C07159=1025.520,281.444,-127.927,170.391,47.586,159.168
C07160=1025.514,281.195,-127.896,170.386,47.588,159.168
C07161=1025.507,280.947,-127.864,170.382,47.590,159.168
C07162=1025.501,280.699,-127.834,170.378,47.592,159.168
C07163=1025.495,280.452,-127.803,170.374,47.594,159.168
C07164=1025.487,280.204,-127.772,170.369,47.596,159.167
C07165=1025.481,279.956,-127.741,170.364,47.598,159.167
C07166=1025.474,279.708,-127.710,170.361,47.600,159.167
C07167=1025.468,279.459,-127.679,170.356,47.602,159.167
C07168=1025.461,279.212,-127.648,170.352,47.604,159.167
C07169=1025.455,278.963,-127.617,170.347,47.606,159.167
C07170=1025.448,278.716,-127.586,170.343,47.608,159.167
C07171=1025.437,278.308,-127.536,170.336,47.611,159.166
C07172=1025.427,277.900,-127.485,170.329,47.615,159.166
C07173=1025.416,277.492,-127.434,170.322,47.618,159.166
C07174=1025.405,277.084,-127.384,170.315,47.621,159.166
C07175=1025.399,276.836,-127.353,170.311,47.623,159.166
C07176=1025.392,276.588,-127.322,170.306,47.625,159.166
C07177=1025.385,276.340,-127.292,170.302,47.627,159.166
C07178=1025.379,276.092,-127.261,170.298,47.630,159.166
C07179=1025.372,275.843,-127.231,170.294,47.632,159.165
C07180=1025.366,275.596,-127.200,170.290,47.634,159.165
C07181=1025.359,275.348,-127.170,170.286,47.636,159.165
C07182=1025.352,275.100,-127.139,170.281,47.638,159.165
C07183=1025.346,274.852,-127.109,170.277,47.640,159.165
C07184=1025.339,274.604,-127.079,170.272,47.642,159.165
C07185=1025.333,274.356,-127.049,170.269,47.645,159.165
C07186=1025.326,274.108,-127.018,170.264,47.647,159.165
C07187=1025.319,273.860,-126.987,170.259,47.649,159.165
C07188=1025.314,273.612,-126.957,170.256,47.651,159.165
C07189=1025.306,273.364,-126.927,170.251,47.653,159.165
C07190=1025.300,273.115,-126.896,170.248,47.655,159.164
C07191=1025.293,272.868,-126.866,170.243,47.658,159.164
C07192=1025.287,272.619,-126.835,170.239,47.659,159.164
C07193=1025.280,272.371,-126.806,170.235,47.662,159.164
C07194=1025.274,272.123,-126.775,170.230,47.664,159.164
C07195=1025.267,271.875,-126.745,170.227,47.666,159.164
C07196=1025.261,271.627,-126.714,170.222,47.669,159.164
C07197=1025.254,271.379,-126.684,170.218,47.670,159.164
C07198=1025.248,271.131,-126.654,170.214,47.673,159.164
C07199=1025.241,270.883,-126.624,170.209,47.675,159.164
C07200=1025.235,270.635,-126.594,170.206,47.678,159.164
C07201=1025.228,270.387,-126.563,170.201,47.680,159.164
C07202=1025.222,270.139,-126.533,170.198,47.682,159.164
C07203=1025.215,269.891,-126.503,170.193,47.684,159.164
C07204=1025.208,269.643,-126.473,170.190,47.687,159.164
C07205=1025.202,269.394,-126.443,170.185,47.689,159.164
C07206=1025.196,269.146,-126.413,170.182,47.691,159.164
C07207=1025.189,268.898,-126.383,170.177,47.693,159.163
C07208=1025.183,268.650,-126.353,170.172,47.696,159.163
C07209=1025.176,268.402,-126.323,170.169,47.698,159.164
C07210=1025.169,268.154,-126.294,170.164,47.700,159.163
C07211=1025.163,267.906,-126.263,170.161,47.703,159.163
C07212=1025.156,267.658,-126.233,170.156,47.705,159.163
C07213=1025.150,267.409,-126.204,170.153,47.707,159.163
C07214=1025.144,267.161,-126.174,170.148,47.710,159.163
C07215=1025.137,266.913,-126.143,170.144,47.712,159.163
C07216=1025.130,266.666,-126.114,170.140,47.715,159.163
C07217=1025.124,266.417,-126.084,170.136,47.717,159.163
C07218=1025.117,266.169,-126.054,170.132,47.719,159.163
C07219=1025.110,265.920,-126.025,170.128,47.722,159.163
C07220=1025.104,265.673,-125.995,170.124,47.724,159.163
C07221=1025.097,265.425,-125.965,170.120,47.727,159.163
C07222=1025.091,265.176,-125.935,170.116,47.729,159.163
C07223=1025.085,264.928,-125.905,170.112,47.731,159.163
C07224=1025.078,264.680,-125.876,170.107,47.734,159.163
C07225=1025.071,264.432,-125.846,170.104,47.737,159.163
C07226=1025.064,264.183,-125.817,170.099,47.739,159.163
C07227=1025.054,263.780,-125.768,170.093,47.743,159.163
C07228=1025.044,263.378,-125.720,170.087,47.747,159.163
C07229=1025.034,262.974,-125.672,170.080,47.751,159.163
C07230=1025.023,262.571,-125.624,170.074,47.755,159.163
C07231=1025.016,262.322,-125.595,170.069,47.757,159.163
C07232=1025.010,262.075,-125.565,170.066,47.760,159.163
C07233=1025.003,261.827,-125.536,170.061,47.763,159.163
C07234=1024.996,261.578,-125.506,170.058,47.765,159.163
C07235=1024.991,261.330,-125.476,170.054,47.768,159.163
C07236=1024.984,261.082,-125.447,170.050,47.770,159.163
C07237=1024.977,260.834,-125.417,170.046,47.773,159.163
C07238=1024.971,260.586,-125.388,170.042,47.775,159.164
C07239=1024.965,260.337,-125.359,170.038,47.778,159.164
C07240=1024.957,260.089,-125.330,170.034,47.781,159.164
C07241=1024.951,259.841,-125.301,170.030,47.783,159.164
C07242=1024.945,259.593,-125.272,170.026,47.786,159.164
C07243=1024.937,259.344,-125.242,170.022,47.788,159.164
C07244=1024.930,259.097,-125.213,170.018,47.791,159.164
C07245=1024.924,258.848,-125.184,170.014,47.794,159.164
C07246=1024.917,258.600,-125.155,170.010,47.796,159.164
C07247=1024.911,258.351,-125.126,170.006,47.800,159.164
C07248=1024.904,258.104,-125.097,170.003,47.802,159.164
C07249=1024.897,257.855,-125.068,169.998,47.805,159.164
C07250=1024.891,257.607,-125.039,169.994,47.807,159.164
C07251=1024.885,257.359,-125.010,169.990,47.810,159.164
C07252=1024.878,257.111,-124.981,169.986,47.813,159.164
C07253=1024.871,256.862,-124.952,169.983,47.816,159.164
C07254=1024.865,256.614,-124.923,169.979,47.818,159.164
C07255=1024.858,256.366,-124.894,169.975,47.821,159.164
C07256=1024.851,256.118,-124.865,169.971,47.824,159.164
C07257=1024.845,255.869,-124.836,169.967,47.826,159.165
C07258=1024.838,255.621,-124.807,169.963,47.829,159.165
C07259=1024.832,255.373,-124.778,169.959,47.832,159.165
C07260=1024.825,255.125,-124.750,169.955,47.835,159.165
C07261=1024.818,254.876,-124.720,169.951,47.837,159.165
C07262=1024.812,254.628,-124.691,169.948,47.840,159.165
C07263=1024.806,254.379,-124.663,169.944,47.843,159.165
C07264=1024.799,254.131,-124.634,169.940,47.846,159.165
C07265=1024.793,253.883,-124.605,169.936,47.848,159.165
C07266=1024.787,253.635,-124.576,169.933,47.851,159.165
C07267=1024.779,253.387,-124.547,169.928,47.854,159.165
C07268=1024.773,253.138,-124.518,169.925,47.857,159.165
C07269=1024.767,252.890,-124.489,169.921,47.860,159.166
C07270=1024.761,252.642,-124.461,169.916,47.863,159.166
C07271=1024.754,252.394,-124.433,169.913,47.865,159.166
C07272=1024.747,252.146,-124.404,169.909,47.869,159.166
C07273=1024.741,251.897,-124.375,169.906,47.871,159.166
C07274=1024.734,251.649,-124.345,169.901,47.874,159.166
C07275=1024.728,251.400,-124.317,169.898,47.877,159.166
C07276=1024.721,251.152,-124.288,169.894,47.880,159.166
C07277=1024.715,250.904,-124.259,169.890,47.882,159.166
C07278=1024.708,250.656,-124.231,169.886,47.885,159.166
C07279=1024.702,250.407,-124.203,169.883,47.888,159.167
C07280=1024.696,250.159,-124.173,169.878,47.891,159.167
C07281=1024.690,249.911,-124.144,169.875,47.894,159.167
C07282=1024.683,249.663,-124.117,169.871,47.896,159.167
C07283=1024.672,249.258,-124.069,169.865,47.901,159.167
C07284=1024.662,248.853,-124.023,169.859,47.906,159.167
C07285=1024.652,248.448,-123.976,169.852,47.911,159.167
C07286=1024.641,248.044,-123.929,169.847,47.915,159.168
C07287=1024.635,247.795,-123.901,169.843,47.919,159.168
C07288=1024.628,247.547,-123.872,169.839,47.921,159.168
C07289=1024.622,247.299,-123.843,169.835,47.924,159.168
C07290=1024.616,247.050,-123.815,169.832,47.927,159.168
C07291=1024.609,246.802,-123.787,169.827,47.930,159.168
C07292=1024.603,246.554,-123.758,169.824,47.933,159.168
C07293=1024.597,246.305,-123.729,169.821,47.935,159.168
C07294=1024.590,246.057,-123.702,169.817,47.939,159.169
C07295=1024.584,245.809,-123.673,169.813,47.941,159.169
C07296=1024.578,245.560,-123.644,169.809,47.944,159.169
C07297=1024.572,245.312,-123.615,169.806,47.947,159.169
C07298=1024.565,245.064,-123.587,169.802,47.950,159.169
C07299=1024.560,244.816,-123.559,169.799,47.953,159.169
C07300=1024.554,244.567,-123.530,169.794,47.956,159.169
C07301=1024.547,244.320,-123.502,169.791,47.959,159.170
C07302=1024.541,244.071,-123.474,169.787,47.962,159.170
C07303=1024.535,243.823,-123.445,169.784,47.965,159.170
C07304=1024.528,243.574,-123.417,169.779,47.968,159.170
C07305=1024.522,243.325,-123.389,169.776,47.971,159.170
C07306=1024.515,243.078,-123.360,169.772,47.974,159.170
C07307=1024.508,242.829,-123.332,169.769,47.977,159.170
C07308=1024.502,242.580,-123.304,169.765,47.980,159.171
C07309=1024.495,242.333,-123.276,169.762,47.983,159.171
C07310=1024.490,242.085,-123.248,169.758,47.987,159.171
C07311=1024.483,241.836,-123.220,169.754,47.989,159.171
C07312=1024.477,241.588,-123.192,169.750,47.993,159.171
C07313=1024.471,241.339,-123.164,169.747,47.996,159.171
C07314=1024.464,241.091,-123.135,169.743,47.999,159.172
C07315=1024.458,240.842,-123.107,169.740,48.002,159.172
C07316=1024.451,240.594,-123.079,169.735,48.005,159.172
C07317=1024.445,240.345,-123.051,169.732,48.008,159.172
C07318=1024.438,240.097,-123.023,169.728,48.011,159.172
C07319=1024.432,239.850,-122.995,169.725,48.015,159.173
C07320=1024.426,239.601,-122.967,169.721,48.017,159.173
C07321=1024.419,239.352,-122.939,169.718,48.020,159.173
C07322=1024.413,239.104,-122.911,169.714,48.024,159.173
C07323=1024.406,238.856,-122.884,169.711,48.027,159.173
C07324=1024.399,238.607,-122.856,169.707,48.030,159.173
C07325=1024.394,238.359,-122.828,169.703,48.033,159.174
C07326=1024.387,238.111,-122.800,169.699,48.037,159.174
C07327=1024.381,237.862,-122.773,169.696,48.040,159.174
C07328=1024.374,237.614,-122.745,169.692,48.043,159.174
C07329=1024.367,237.365,-122.717,169.688,48.047,159.174
C07330=1024.361,237.117,-122.689,169.685,48.050,159.175
C07331=1024.355,236.869,-122.661,169.681,48.053,159.175
C07332=1024.349,236.620,-122.634,169.678,48.056,159.175
C07333=1024.342,236.372,-122.606,169.674,48.060,159.175
C07334=1024.336,236.123,-122.579,169.671,48.063,159.176
C07335=1024.329,235.874,-122.551,169.667,48.066,159.176
C07336=1024.323,235.627,-122.524,169.664,48.070,159.176
C07337=1024.316,235.378,-122.496,169.660,48.073,159.176
C07338=1024.309,235.130,-122.468,169.657,48.076,159.176
C07339=1024.299,234.719,-122.423,169.650,48.082,159.177
C07340=1024.288,234.308,-122.377,169.645,48.087,159.177
C07341=1024.277,233.897,-122.332,169.638,48.093,159.177
C07342=1024.267,233.486,-122.286,169.633,48.098,159.178
C07343=1024.260,233.238,-122.259,169.629,48.101,159.178
C07344=1024.255,232.988,-122.231,169.626,48.104,159.178
C07345=1024.248,232.740,-122.203,169.622,48.108,159.179
C07346=1024.242,232.492,-122.176,169.619,48.112,159.179
C07347=1024.235,232.244,-122.148,169.615,48.115,159.179
C07348=1024.229,231.995,-122.121,169.612,48.118,159.179
C07349=1024.223,231.747,-122.094,169.608,48.122,159.179
C07350=1024.216,231.499,-122.066,169.604,48.125,159.180
C07351=1024.210,231.249,-122.039,169.600,48.128,159.180
C07352=1024.204,231.002,-122.012,169.598,48.132,159.180
C07353=1024.197,230.753,-121.984,169.594,48.135,159.180
C07354=1024.190,230.505,-121.956,169.591,48.138,159.181
C07355=1024.185,230.256,-121.929,169.586,48.142,159.181
C07356=1024.178,230.008,-121.902,169.583,48.145,159.181
C07357=1024.172,229.759,-121.875,169.580,48.149,159.181
C07358=1024.165,229.511,-121.847,169.577,48.152,159.182
C07359=1024.159,229.262,-121.820,169.573,48.156,159.182
C07360=1024.152,229.014,-121.793,169.569,48.159,159.182
C07361=1024.146,228.766,-121.765,169.566,48.163,159.182
C07362=1024.140,228.517,-121.738,169.562,48.166,159.183
C07363=1024.133,228.268,-121.711,169.559,48.169,159.183
C07364=1024.127,228.020,-121.684,169.555,48.173,159.183
C07365=1024.120,227.772,-121.657,169.552,48.177,159.183
C07366=1024.114,227.523,-121.630,169.548,48.180,159.184
C07367=1024.108,227.275,-121.602,169.545,48.184,159.184
C07368=1024.101,227.026,-121.575,169.541,48.187,159.184
C07369=1024.095,226.778,-121.549,169.538,48.190,159.184
C07370=1024.088,226.530,-121.522,169.534,48.194,159.185
C07371=1024.082,226.281,-121.495,169.531,48.198,159.185
C07372=1024.076,226.033,-121.467,169.527,48.202,159.185
C07373=1024.068,225.784,-121.441,169.524,48.205,159.186
C07374=1024.063,225.536,-121.414,169.520,48.209,159.186
C07375=1024.056,225.287,-121.386,169.516,48.212,159.186
C07376=1024.049,225.039,-121.360,169.514,48.216,159.187
C07377=1024.043,224.790,-121.333,169.510,48.220,159.187
C07378=1024.037,224.541,-121.306,169.507,48.223,159.187
C07379=1024.031,224.293,-121.279,169.503,48.227,159.187
C07380=1024.024,224.045,-121.253,169.500,48.231,159.188
C07381=1024.018,223.796,-121.226,169.496,48.234,159.188
C07382=1024.011,223.547,-121.199,169.493,48.238,159.188
C07383=1024.004,223.299,-121.172,169.489,48.241,159.189
C07384=1023.998,223.051,-121.145,169.486,48.245,159.189
C07385=1023.992,222.802,-121.118,169.482,48.248,159.189
C07386=1023.985,222.554,-121.092,169.479,48.253,159.190
C07387=1023.979,222.305,-121.064,169.476,48.256,159.190
C07388=1023.973,222.057,-121.038,169.472,48.260,159.190
C07389=1023.966,221.808,-121.011,169.469,48.263,159.190
C07390=1023.960,221.560,-120.985,169.465,48.267,159.191
C07391=1023.954,221.311,-120.958,169.462,48.271,159.191
C07392=1023.947,221.063,-120.931,169.458,48.274,159.191
C07393=1023.940,220.814,-120.904,169.456,48.278,159.192
C07394=1023.935,220.566,-120.877,169.451,48.282,159.192
C07395=1023.924,220.147,-120.832,169.446,48.288,159.192
C07396=1023.913,219.728,-120.787,169.441,48.294,159.193
C07397=1023.902,219.309,-120.742,169.434,48.301,159.194
C07398=1023.892,218.890,-120.698,169.429,48.307,159.194
C07399=1023.885,218.641,-120.671,169.426,48.311,159.195
C07400=1023.879,218.393,-120.645,169.422,48.314,159.195
C07401=1023.872,218.144,-120.618,169.419,48.318,159.195
C07402=1023.866,217.896,-120.592,169.415,48.322,159.195
C07403=1023.859,217.648,-120.566,169.412,48.326,159.196
C07404=1023.852,217.399,-120.539,169.408,48.329,159.196
C07405=1023.847,217.151,-120.513,169.406,48.333,159.196
C07406=1023.839,216.902,-120.486,169.402,48.337,159.197
C07407=1023.834,216.654,-120.460,169.398,48.342,159.197
C07408=1023.827,216.405,-120.433,169.395,48.345,159.198
C07409=1023.820,216.157,-120.407,169.392,48.349,159.198
C07410=1023.814,215.909,-120.380,169.389,48.353,159.198
C07411=1023.808,215.659,-120.355,169.385,48.357,159.199
C07412=1023.801,215.411,-120.329,169.382,48.361,159.199
C07413=1023.795,215.162,-120.302,169.378,48.365,159.199
C07414=1023.788,214.914,-120.276,169.375,48.369,159.200
C07415=1023.782,214.666,-120.249,169.372,48.373,159.200
C07416=1023.775,214.417,-120.223,169.368,48.377,159.200
C07417=1023.769,214.168,-120.197,169.365,48.380,159.201
C07418=1023.763,213.919,-120.170,169.362,48.384,159.201
C07419=1023.756,213.671,-120.144,169.359,48.388,159.201
C07420=1023.750,213.423,-120.118,169.355,48.392,159.202
C07421=1023.743,213.174,-120.091,169.351,48.396,159.202
C07422=1023.737,212.925,-120.066,169.349,48.400,159.203
C07423=1023.731,212.677,-120.040,169.345,48.404,159.203
C07424=1023.724,212.428,-120.013,169.342,48.408,159.203
C07425=1023.718,212.180,-119.987,169.338,48.412,159.204
C07426=1023.712,211.931,-119.961,169.336,48.416,159.204
C07427=1023.705,211.682,-119.934,169.332,48.420,159.204
C07428=1023.699,211.434,-119.908,169.329,48.424,159.205
C07429=1023.693,211.185,-119.882,169.326,48.428,159.205
C07430=1023.686,210.937,-119.856,169.321,48.431,159.205
C07431=1023.679,210.689,-119.830,169.319,48.435,159.206
C07432=1023.674,210.440,-119.804,169.315,48.439,159.206
C07433=1023.667,210.192,-119.778,169.312,48.443,159.207
C07434=1023.660,209.943,-119.751,169.309,48.448,159.207
C07435=1023.654,209.694,-119.726,169.306,48.452,159.208
C07436=1023.648,209.446,-119.700,169.303,48.456,159.208
C07437=1023.642,209.196,-119.674,169.299,48.460,159.208
C07438=1023.635,208.948,-119.648,169.296,48.464,159.209
C07439=1023.629,208.700,-119.622,169.292,48.468,159.209
C07440=1023.622,208.452,-119.596,169.290,48.472,159.209
C07441=1023.615,208.203,-119.570,169.286,48.476,159.210
C07442=1023.609,207.954,-119.544,169.282,48.480,159.210
C07443=1023.603,207.706,-119.518,169.279,48.484,159.211
C07444=1023.597,207.457,-119.492,169.276,48.488,159.211
C07445=1023.590,207.208,-119.466,169.273,48.492,159.212
C07446=1023.584,206.960,-119.441,169.270,48.496,159.212
C07447=1023.577,206.712,-119.415,169.266,48.501,159.212
C07448=1023.571,206.463,-119.389,169.263,48.504,159.213
C07449=1023.564,206.214,-119.364,169.260,48.509,159.213
C07450=1023.558,205.966,-119.338,169.257,48.513,159.214
C07451=1023.547,205.550,-119.295,169.251,48.520,159.214
C07452=1023.536,205.133,-119.251,169.246,48.527,159.215
C07453=1023.525,204.716,-119.209,169.240,48.534,159.216
C07454=1023.515,204.300,-119.166,169.236,48.541,159.216
C07455=1023.491,203.269,-119.066,168.819,48.442,159.136
C07456=1023.486,203.020,-119.041,168.815,48.447,159.136
C07457=1023.480,202.772,-119.017,168.811,48.452,159.136
C07458=1023.474,202.523,-118.993,168.806,48.457,159.137
C07459=1023.469,202.274,-118.969,168.802,48.463,159.137
C07460=1023.464,202.025,-118.945,168.798,48.468,159.138
C07461=1023.458,201.776,-118.921,168.794,48.472,159.138
C07462=1023.452,201.528,-118.897,168.790,48.478,159.139
C07463=1023.446,201.279,-118.873,168.786,48.483,159.139
C07464=1023.441,201.030,-118.848,168.781,48.488,159.140
C07465=1023.436,200.781,-118.825,168.778,48.493,159.140
C07466=1023.429,200.532,-118.801,168.773,48.498,159.141
C07467=1023.424,200.284,-118.777,168.769,48.503,159.141
C07468=1023.419,200.035,-118.752,168.764,48.509,159.141
C07469=1023.413,199.786,-118.728,168.761,48.513,159.142
C07470=1023.407,199.537,-118.705,168.757,48.518,159.142
C07471=1023.402,199.288,-118.681,168.753,48.524,159.143
C07472=1023.396,199.039,-118.658,168.748,48.529,159.143
C07473=1023.390,198.791,-118.634,168.744,48.534,159.144
C07474=1023.385,198.542,-118.610,168.740,48.539,159.144
C07475=1023.378,198.293,-118.586,168.736,48.545,159.145
C07476=1023.372,198.045,-118.563,168.732,48.550,159.145
C07477=1023.367,197.795,-118.539,168.727,48.555,159.146
C07478=1023.361,197.547,-118.515,168.724,48.561,159.146
C07479=1023.356,197.298,-118.492,168.720,48.566,159.147
C07480=1023.350,197.049,-118.468,168.715,48.571,159.147
C07481=1023.344,196.800,-118.445,168.711,48.576,159.148
C07482=1023.339,196.551,-118.421,168.708,48.582,159.148
C07483=1023.333,196.303,-118.398,168.703,48.587,159.149
C07484=1023.328,196.054,-118.374,168.699,48.592,159.149
C07485=1023.322,195.805,-118.351,168.695,48.598,159.150
C07486=1023.316,195.557,-118.327,168.692,48.602,159.150
C07487=1023.310,195.307,-118.303,168.687,48.608,159.151
C07488=1023.305,195.058,-118.280,168.683,48.613,159.151
C07489=1023.299,194.810,-118.256,168.679,48.619,159.152
C07490=1023.294,194.560,-118.233,168.675,48.623,159.152
C07491=1023.288,194.312,-118.209,168.671,48.628,159.152
C07492=1023.283,194.063,-118.186,168.667,48.634,159.153
C07493=1023.277,193.814,-118.163,168.663,48.639,159.154
C07494=1023.271,193.566,-118.139,168.659,48.644,159.154
C07495=1023.266,193.317,-118.116,168.655,48.650,159.155
C07496=1023.260,193.068,-118.092,168.651,48.655,159.155
C07497=1023.254,192.819,-118.069,168.647,48.660,159.155
C07498=1023.249,192.570,-118.045,168.643,48.666,159.156
C07499=1023.243,192.321,-118.022,168.640,48.671,159.157
C07500=1023.238,192.073,-117.998,168.635,48.676,159.157
C07501=1023.232,191.824,-117.975,168.631,48.682,159.158
C07502=1023.227,191.575,-117.952,168.628,48.686,159.158
C07503=1023.221,191.326,-117.928,168.623,48.692,159.158
C07504=1023.215,191.077,-117.905,168.619,48.697,159.159
C07505=1023.210,190.829,-117.882,168.616,48.702,159.160
C07506=1023.205,190.579,-117.859,168.611,48.707,159.160
C07507=1023.199,190.331,-117.835,168.607,48.713,159.161
C07508=1023.193,190.082,-117.812,168.604,48.718,159.161
C07509=1023.188,189.833,-117.788,168.600,48.724,159.162
C07510=1023.182,189.584,-117.765,168.595,48.729,159.162
C07511=1023.177,189.336,-117.741,168.592,48.734,159.163
C07512=1023.171,189.087,-117.718,168.588,48.740,159.163
C07513=1023.166,188.838,-117.695,168.584,48.744,159.164
C07514=1023.161,188.588,-117.672,168.580,48.750,159.164
C07515=1023.155,188.340,-117.649,168.576,48.755,159.165
C07516=1023.148,188.058,-117.622,168.572,48.761,159.165
C07517=1023.142,187.776,-117.596,168.568,48.767,159.166
C07518=1023.136,187.494,-117.570,168.563,48.773,159.166
C07519=1023.131,187.212,-117.543,168.559,48.779,159.167
C07520=1023.125,186.963,-117.521,168.555,48.784,159.167
C07521=1023.119,186.714,-117.498,168.551,48.790,159.168
C07522=1023.114,186.465,-117.474,168.547,48.795,159.168
C07523=1023.108,186.216,-117.451,168.543,48.800,159.169
C07524=1023.102,185.967,-117.427,168.539,48.806,159.169
C07525=1023.097,185.718,-117.404,168.536,48.810,159.170
C07526=1023.092,185.469,-117.381,168.532,48.816,159.171
C07527=1023.087,185.221,-117.358,168.529,48.821,159.171
C07528=1023.082,184.972,-117.335,168.524,48.826,159.171
C07529=1023.076,184.723,-117.312,168.521,48.832,159.172
C07530=1023.070,184.474,-117.289,168.517,48.837,159.173
C07531=1023.065,184.225,-117.265,168.513,48.842,159.173
C07532=1023.059,183.976,-117.242,168.509,48.848,159.174
C07533=1023.054,183.728,-117.220,168.506,48.853,159.174
C07534=1023.049,183.479,-117.196,168.502,48.858,159.175
C07535=1023.044,183.230,-117.173,168.498,48.863,159.175
C07536=1023.038,182.981,-117.150,168.494,48.868,159.176
C07537=1023.033,182.731,-117.128,168.491,48.874,159.176
C07538=1023.027,182.482,-117.105,168.487,48.879,159.177
C07539=1023.022,182.234,-117.082,168.484,48.885,159.177
C07540=1023.017,181.985,-117.059,168.479,48.890,159.178
C07541=1023.011,181.735,-117.037,168.475,48.896,159.178
C07542=1023.005,181.487,-117.015,168.472,48.901,159.179
C07543=1022.999,181.238,-116.992,168.468,48.907,159.180
C07544=1022.993,180.988,-116.969,168.464,48.912,159.180
C07545=1022.988,180.741,-116.947,168.461,48.918,159.181
C07546=1022.982,180.491,-116.925,168.457,48.924,159.181
C07547=1022.976,180.242,-116.902,168.453,48.929,159.182
C07548=1022.971,179.993,-116.879,168.449,48.934,159.182
C07549=1022.965,179.744,-116.858,168.445,48.940,159.183
C07550=1022.959,179.495,-116.835,168.442,48.946,159.184
C07551=1022.954,179.246,-116.813,168.438,48.951,159.184
C07552=1022.948,178.998,-116.790,168.435,48.957,159.185
C07553=1022.942,178.748,-116.768,168.431,48.962,159.185
C07554=1022.936,178.499,-116.745,168.426,48.968,159.186
C07555=1022.931,178.251,-116.724,168.423,48.973,159.186
C07556=1022.925,178.002,-116.701,168.419,48.979,159.187
C07557=1022.920,177.752,-116.679,168.416,48.985,159.188
C07558=1022.914,177.504,-116.656,168.412,48.990,159.188
C07559=1022.908,177.255,-116.635,168.409,48.995,159.189
C07560=1022.903,177.006,-116.612,168.405,49.001,159.189
C07561=1022.897,176.757,-116.589,168.401,49.006,159.190
C07562=1022.891,176.508,-116.567,168.397,49.012,159.190
C07563=1022.886,176.259,-116.545,168.393,49.018,159.191
C07564=1022.880,176.010,-116.522,168.390,49.023,159.192
C07565=1022.874,175.761,-116.501,168.386,49.029,159.192
C07566=1022.869,175.513,-116.478,168.383,49.034,159.193
C07567=1022.863,175.263,-116.456,168.379,49.040,159.193
C07568=1022.858,175.014,-116.434,168.376,49.046,159.194
C07569=1022.852,174.766,-116.412,168.371,49.051,159.194
C07570=1022.847,174.516,-116.389,168.368,49.056,159.195
C07571=1022.841,174.268,-116.366,168.364,49.062,159.195
C07572=1022.835,174.019,-116.345,168.361,49.068,159.196
C07573=1022.830,173.770,-116.323,168.357,49.073,159.197
C07574=1022.824,173.521,-116.300,168.354,49.079,159.197
C07575=1022.819,173.272,-116.279,168.350,49.084,159.198
C07576=1022.813,173.023,-116.257,168.346,49.089,159.198
C07577=1022.808,172.774,-116.234,168.342,49.095,159.199
C07578=1022.802,172.525,-116.212,168.339,49.101,159.200
C07579=1022.797,172.276,-116.190,168.335,49.107,159.200
C07580=1022.791,171.993,-116.164,168.331,49.113,159.201
C07581=1022.784,171.711,-116.140,168.328,49.119,159.201
C07582=1022.778,171.428,-116.114,168.324,49.125,159.202
C07583=1022.771,171.146,-116.089,168.320,49.132,159.203
C07584=1022.766,170.897,-116.067,168.315,49.137,159.203
C07585=1022.760,170.648,-116.046,168.312,49.142,159.204
C07586=1022.755,170.399,-116.024,168.308,49.148,159.204
C07587=1022.750,170.150,-116.001,168.305,49.154,159.205
C07588=1022.744,169.901,-115.979,168.301,49.159,159.206
C07589=1022.739,169.652,-115.958,168.298,49.165,159.206
C07590=1022.734,169.403,-115.935,168.295,49.170,159.207
C07591=1022.728,169.154,-115.914,168.291,49.176,159.207
C07592=1022.722,168.905,-115.891,168.288,49.181,159.208
C07593=1022.717,168.657,-115.869,168.284,49.187,159.208
C07594=1022.711,168.407,-115.848,168.281,49.192,159.209
C07595=1022.706,168.158,-115.825,168.277,49.197,159.210
C07596=1022.701,167.909,-115.803,168.273,49.203,159.210
C07597=1022.695,167.660,-115.782,168.270,49.209,159.211
C07598=1022.690,167.412,-115.759,168.266,49.215,159.211
C07599=1022.684,167.162,-115.737,168.263,49.220,159.212
C07600=1022.679,166.914,-115.716,168.260,49.225,159.213
C07601=1022.674,166.665,-115.694,168.256,49.231,159.213
C07602=1022.668,166.415,-115.672,168.253,49.237,159.214
C07603=1022.663,166.167,-115.650,168.250,49.242,159.214
C07604=1022.657,165.917,-115.628,168.246,49.248,159.215
C07605=1022.653,165.669,-115.606,168.243,49.253,159.216
C07606=1022.646,165.419,-115.585,168.240,49.259,159.216
C07607=1022.642,165.170,-115.563,168.235,49.264,159.217
C07608=1022.636,164.922,-115.540,168.232,49.270,159.217
C07609=1022.630,164.673,-115.519,168.228,49.276,159.218
C07610=1022.625,164.424,-115.496,168.225,49.280,159.218
C07611=1022.620,164.175,-115.475,168.222,49.286,159.219
C07612=1022.615,163.926,-115.453,168.218,49.292,159.220
C07613=1022.609,163.677,-115.431,168.215,49.298,159.220
C07614=1022.604,163.428,-115.409,168.211,49.303,159.221
C07615=1022.598,163.179,-115.388,168.209,49.308,159.221
C07616=1022.593,162.930,-115.366,168.204,49.314,159.222
C07617=1022.588,162.681,-115.344,168.201,49.319,159.222
C07618=1022.582,162.432,-115.322,168.198,49.325,159.223
C07619=1022.578,162.183,-115.300,168.194,49.331,159.224
C07620=1022.572,161.934,-115.278,168.191,49.336,159.224
C07621=1022.567,161.684,-115.257,168.188,49.341,159.225
C07622=1022.562,161.436,-115.236,168.184,49.347,159.225
C07623=1022.556,161.186,-115.214,168.181,49.353,159.226
C07624=1022.551,160.938,-115.192,168.178,49.358,159.227
C07625=1022.546,160.689,-115.170,168.175,49.363,159.227
C07626=1022.540,160.440,-115.149,168.171,49.369,159.228
C07627=1022.535,160.191,-115.127,168.168,49.375,159.228
C07628=1022.530,159.942,-115.105,168.164,49.380,159.229
C07629=1022.524,159.693,-115.083,168.161,49.385,159.230
C07630=1022.519,159.444,-115.061,168.157,49.391,159.230
C07631=1022.515,159.194,-115.040,168.154,49.397,159.231
C07632=1022.509,158.945,-115.019,168.151,49.402,159.231
C07633=1022.503,158.697,-114.997,168.147,49.408,159.232
C07634=1022.498,158.448,-114.976,168.144,49.413,159.233
C07635=1022.492,158.198,-114.955,168.141,49.419,159.233
C07636=1022.487,157.950,-114.933,168.137,49.425,159.234
C07637=1022.482,157.700,-114.913,168.134,49.431,159.234
C07638=1022.475,157.451,-114.891,168.131,49.436,159.235
C07639=1022.470,157.203,-114.870,168.127,49.442,159.236
C07640=1022.465,156.953,-114.849,168.124,49.448,159.236
C07641=1022.459,156.704,-114.827,168.121,49.453,159.237
C07642=1022.454,156.456,-114.806,168.117,49.459,159.238
C07643=1022.448,156.207,-114.785,168.114,49.465,159.238
C07644=1022.442,155.924,-114.761,168.110,49.471,159.239
C07645=1022.436,155.640,-114.737,168.106,49.477,159.240
C07646=1022.429,155.358,-114.713,168.103,49.484,159.240
C07647=1022.423,155.075,-114.689,168.099,49.491,159.241
C07648=1022.418,154.826,-114.668,168.096,49.496,159.242
C07649=1022.413,154.577,-114.646,168.092,49.502,159.242
C07650=1022.407,154.327,-114.625,168.089,49.507,159.243
C07651=1022.402,154.079,-114.604,168.086,49.513,159.243
C07652=1022.396,153.830,-114.583,168.082,49.519,159.244
C07653=1022.390,153.580,-114.562,168.079,49.525,159.245
C07654=1022.385,153.331,-114.541,168.076,49.530,159.245
C07655=1022.380,153.083,-114.519,168.073,49.536,159.246
C07656=1022.375,152.833,-114.499,168.069,49.542,159.247
C07657=1022.369,152.584,-114.478,168.066,49.547,159.247
C07658=1022.363,152.335,-114.457,168.063,49.553,159.248
C07659=1022.358,152.086,-114.436,168.059,49.559,159.249
C07660=1022.353,151.837,-114.415,168.056,49.565,159.249
C07661=1022.347,151.588,-114.394,168.053,49.570,159.250
C07662=1022.341,151.338,-114.373,168.049,49.576,159.250
C07663=1022.336,151.090,-114.352,168.046,49.582,159.251
C07664=1022.331,150.841,-114.331,168.043,49.588,159.252
C07665=1022.325,150.592,-114.311,168.040,49.593,159.252
C07666=1022.319,150.343,-114.289,168.036,49.599,159.253
C07667=1022.314,150.093,-114.269,168.034,49.605,159.254
C07668=1022.309,149.844,-114.248,168.031,49.611,159.254
C07669=1022.303,149.596,-114.227,168.028,49.616,159.255
C07670=1022.298,149.347,-114.206,168.024,49.622,159.256
C07671=1022.292,149.097,-114.185,168.021,49.628,159.256
C07672=1022.286,148.848,-114.164,168.018,49.633,159.257
C07673=1022.281,148.599,-114.144,168.014,49.639,159.257
C07674=1022.276,148.350,-114.123,168.011,49.645,159.258
C07675=1022.271,148.101,-114.103,168.008,49.651,159.259
C07676=1022.265,147.852,-114.081,168.005,49.656,159.259
C07677=1022.259,147.603,-114.060,168.001,49.662,159.260
C07678=1022.254,147.353,-114.040,167.998,49.668,159.261
C07679=1022.249,147.104,-114.019,167.995,49.674,159.261
C07680=1022.243,146.856,-113.998,167.992,49.679,159.262
C07681=1022.238,146.607,-113.977,167.988,49.685,159.263
C07682=1022.232,146.358,-113.957,167.985,49.691,159.263
C07683=1022.226,146.108,-113.937,167.982,49.697,159.264
C07684=1022.221,145.859,-113.916,167.979,49.702,159.265
C07685=1022.216,145.610,-113.895,167.975,49.708,159.265
C07686=1022.210,145.361,-113.875,167.972,49.714,159.266
C07687=1022.205,145.112,-113.854,167.970,49.720,159.267
C07688=1022.199,144.863,-113.834,167.967,49.726,159.267
C07689=1022.194,144.614,-113.813,167.963,49.732,159.268
C07690=1022.188,144.364,-113.792,167.960,49.738,159.268
C07691=1022.182,144.115,-113.772,167.957,49.743,159.269
C07692=1022.176,143.867,-113.752,167.954,49.749,159.270
C07693=1022.171,143.617,-113.731,167.950,49.755,159.270
C07694=1022.166,143.368,-113.711,167.947,49.761,159.271
C07695=1022.161,143.119,-113.690,167.944,49.766,159.272
C07696=1022.155,142.870,-113.670,167.941,49.772,159.272
C07697=1022.149,142.621,-113.649,167.937,49.778,159.273
C07698=1022.144,142.372,-113.629,167.935,49.784,159.274
C07699=1022.138,142.123,-113.609,167.932,49.790,159.274
C07700=1022.133,141.874,-113.588,167.929,49.796,159.275
C07701=1022.127,141.624,-113.567,167.926,49.801,159.276
C07702=1022.122,141.375,-113.547,167.922,49.807,159.276
C07703=1022.116,141.126,-113.527,167.919,49.813,159.277
C07704=1022.111,140.877,-113.506,167.916,49.819,159.278
C07705=1022.105,140.628,-113.486,167.913,49.825,159.278
C07706=1022.100,140.379,-113.465,167.909,49.831,159.279
C07707=1022.094,140.130,-113.446,167.906,49.836,159.280
C07708=1022.089,139.893,-113.426,167.904,49.842,159.280
C07709=1022.084,139.654,-113.407,167.901,49.848,159.281
C07710=1022.079,139.416,-113.387,167.898,49.853,159.282
C07711=1022.074,139.177,-113.368,167.894,49.858,159.282
C07712=1022.069,138.940,-113.348,167.891,49.864,159.283
C07713=1022.064,138.701,-113.329,167.890,49.869,159.283
C07714=1022.058,138.463,-113.309,167.887,49.875,159.284
C07715=1022.053,138.225,-113.291,167.884,49.881,159.285
C07716=1022.047,137.919,-113.265,167.879,49.888,159.285
C07717=1022.040,137.615,-113.240,167.876,49.895,159.286
C07718=1022.033,137.310,-113.216,167.871,49.902,159.287
C07719=1022.026,137.004,-113.191,167.868,49.910,159.288
C07720=1022.020,136.755,-113.171,167.865,49.915,159.289
C07721=1022.015,136.506,-113.151,167.862,49.921,159.289
C07722=1022.009,136.257,-113.131,167.859,49.927,159.290
C07723=1022.004,136.007,-113.111,167.855,49.933,159.290
C07724=1021.998,135.759,-113.091,167.853,49.938,159.291
C07725=1021.993,135.509,-113.071,167.850,49.944,159.292
C07726=1021.987,135.260,-113.051,167.847,49.950,159.293
C07727=1021.982,135.012,-113.031,167.844,49.956,159.293
C07728=1021.977,134.762,-113.012,167.840,49.962,159.294
C07729=1021.971,134.513,-112.991,167.837,49.968,159.295
C07730=1021.965,134.264,-112.971,167.834,49.974,159.295
C07731=1021.960,134.015,-112.951,167.831,49.979,159.296
C07732=1021.954,133.766,-112.931,167.829,49.985,159.296
C07733=1021.949,133.517,-112.911,167.825,49.992,159.297
C07734=1021.943,133.267,-112.892,167.822,49.997,159.298
C07735=1021.938,133.018,-112.871,167.819,50.003,159.299
C07736=1021.932,132.769,-112.851,167.816,50.009,159.299
C07737=1021.927,132.519,-112.831,167.813,50.015,159.300
C07738=1021.921,132.271,-112.811,167.810,50.020,159.301
C07739=1021.916,132.021,-112.792,167.807,50.026,159.301
C07740=1021.910,131.772,-112.772,167.804,50.033,159.302
C07741=1021.905,131.524,-112.752,167.801,50.038,159.303
C07742=1021.900,131.274,-112.732,167.798,50.044,159.303
C07743=1021.894,131.025,-112.712,167.795,50.050,159.304
C07744=1021.889,130.776,-112.692,167.792,50.056,159.305
C07745=1021.883,130.527,-112.672,167.790,50.061,159.305
C07746=1021.878,130.277,-112.653,167.786,50.067,159.306
C07747=1021.872,130.028,-112.633,167.783,50.073,159.306
C07748=1021.866,129.779,-112.613,167.780,50.079,159.307
C07749=1021.861,129.530,-112.593,167.777,50.085,159.308
C07750=1021.856,129.281,-112.574,167.774,50.091,159.309
C07751=1021.850,129.032,-112.555,167.771,50.098,159.309
C07752=1021.844,128.783,-112.535,167.768,50.103,159.310
C07753=1021.839,128.533,-112.515,167.765,50.109,159.311
C07754=1021.833,128.284,-112.496,167.762,50.115,159.311
C07755=1021.827,128.035,-112.476,167.760,50.121,159.312
C07756=1021.821,127.786,-112.457,167.756,50.127,159.313
C07757=1021.816,127.536,-112.437,167.753,50.133,159.313
C07758=1021.810,127.287,-112.417,167.750,50.139,159.314
C07759=1021.805,127.038,-112.398,167.747,50.145,159.315
C07760=1021.800,126.789,-112.379,167.745,50.151,159.316
C07761=1021.794,126.540,-112.359,167.741,50.157,159.316
C07762=1021.788,126.291,-112.340,167.738,50.163,159.317
C07763=1021.782,126.041,-112.321,167.735,50.169,159.318
C07764=1021.776,125.792,-112.301,167.732,50.175,159.318
C07765=1021.771,125.544,-112.282,167.729,50.181,159.319
C07766=1021.766,125.294,-112.262,167.726,50.187,159.320
C07767=1021.761,125.045,-112.243,167.723,50.193,159.320
C07768=1021.755,124.796,-112.223,167.720,50.199,159.321
C07769=1021.749,124.546,-112.204,167.717,50.205,159.322
C07770=1021.744,124.298,-112.185,167.715,50.211,159.323
C07771=1021.738,124.048,-112.165,167.712,50.217,159.323
C07772=1021.732,123.765,-112.143,167.708,50.223,159.324
C07773=1021.726,123.482,-112.121,167.705,50.230,159.325
C07774=1021.719,123.198,-112.099,167.701,50.237,159.325
C07775=1021.713,122.915,-112.077,167.698,50.244,159.326
C07776=1021.707,122.666,-112.058,167.695,50.249,159.327
C07777=1021.701,122.417,-112.038,167.692,50.256,159.328
C07778=1021.696,122.168,-112.019,167.690,50.262,159.328
C07779=1021.691,121.919,-112.000,167.687,50.267,159.329
C07780=1021.685,121.669,-111.980,167.684,50.273,159.330
C07781=1021.679,121.420,-111.961,167.681,50.279,159.330
C07782=1021.674,121.171,-111.942,167.677,50.286,159.331
C07783=1021.668,120.922,-111.922,167.675,50.291,159.332
C07784=1021.662,120.673,-111.903,167.672,50.297,159.332
C07785=1021.658,120.424,-111.883,167.669,50.303,159.333
C07786=1021.652,120.174,-111.864,167.666,50.309,159.334
C07787=1021.647,119.925,-111.845,167.663,50.315,159.335
C07788=1021.641,119.675,-111.826,167.661,50.321,159.335
C07789=1021.636,119.427,-111.807,167.658,50.327,159.336
C07790=1021.630,119.177,-111.788,167.655,50.332,159.337
C07791=1021.624,118.928,-111.768,167.652,50.338,159.337
C07792=1021.619,118.680,-111.749,167.648,50.344,159.338
C07793=1021.614,118.430,-111.730,167.646,50.351,159.339
C07794=1021.608,118.181,-111.710,167.643,50.356,159.339
C07795=1021.603,117.931,-111.690,167.640,50.362,159.340
C07796=1021.598,117.682,-111.672,167.637,50.368,159.341
C07797=1021.592,117.433,-111.652,167.634,50.374,159.341
C07798=1021.586,117.183,-111.633,167.631,50.379,159.342
C07799=1021.581,116.935,-111.614,167.629,50.386,159.343
C07800=1021.576,116.685,-111.595,167.626,50.392,159.343
C07801=1021.570,116.436,-111.576,167.623,50.397,159.344
C07802=1021.565,116.187,-111.557,167.620,50.403,159.345
C07803=1021.559,115.938,-111.538,167.617,50.409,159.345
C07804=1021.554,115.689,-111.519,167.615,50.415,159.346
C07805=1021.548,115.440,-111.499,167.612,50.421,159.347
C07806=1021.543,115.190,-111.480,167.609,50.426,159.347
C07807=1021.538,114.941,-111.461,167.606,50.433,159.348
C07808=1021.533,114.692,-111.442,167.604,50.439,159.349
C07809=1021.527,114.442,-111.422,167.601,50.444,159.349
C07810=1021.522,114.193,-111.403,167.598,50.450,159.350
C07811=1021.516,113.944,-111.384,167.595,50.456,159.351
C07812=1021.511,113.695,-111.365,167.592,50.462,159.351
C07813=1021.505,113.446,-111.346,167.588,50.468,159.352
C07814=1021.500,113.196,-111.327,167.585,50.474,159.353
C07815=1021.495,112.948,-111.308,167.583,50.479,159.353
C07816=1021.489,112.698,-111.289,167.580,50.485,159.354
C07817=1021.483,112.449,-111.269,167.577,50.492,159.355
C07818=1021.479,112.200,-111.251,167.574,50.497,159.355
C07819=1021.473,111.950,-111.232,167.572,50.503,159.356
C07820=1021.468,111.701,-111.213,167.569,50.509,159.357
C07821=1021.462,111.452,-111.194,167.566,50.515,159.357
C07822=1021.456,111.203,-111.175,167.563,50.521,159.358
C07823=1021.451,110.953,-111.157,167.561,50.527,159.359
C07824=1021.445,110.704,-111.138,167.558,50.533,159.360
C07825=1021.440,110.455,-111.119,167.555,50.539,159.360
C07826=1021.434,110.206,-111.100,167.552,50.545,159.361
C07827=1021.428,109.956,-111.082,167.550,50.551,159.362
C07828=1021.423,109.707,-111.063,167.547,50.557,159.362
C07829=1021.417,109.458,-111.044,167.544,50.562,159.363
C07830=1021.412,109.209,-111.026,167.540,50.569,159.364
C07831=1021.406,108.959,-111.007,167.538,50.575,159.364
C07832=1021.401,108.711,-110.988,167.535,50.581,159.365
C07833=1021.395,108.461,-110.970,167.532,50.587,159.366
C07834=1021.389,108.212,-110.951,167.529,50.593,159.367
C07835=1021.385,107.962,-110.933,167.527,50.599,159.367
C07836=1021.378,107.680,-110.911,167.523,50.606,159.368
C07837=1021.372,107.396,-110.891,167.520,50.612,159.369
C07838=1021.365,107.112,-110.870,167.517,50.619,159.370
C07839=1021.359,106.829,-110.848,167.514,50.626,159.371
C07840=1021.353,106.580,-110.830,167.511,50.632,159.371
C07841=1021.347,106.331,-110.811,167.509,50.638,159.372
C07842=1021.343,106.082,-110.793,167.506,50.644,159.373
C07843=1021.336,105.832,-110.774,167.503,50.650,159.373
C07844=1021.331,105.584,-110.755,167.499,50.656,159.374
C07845=1021.325,105.334,-110.737,167.497,50.662,159.375
C07846=1021.320,105.085,-110.718,167.494,50.668,159.375
C07847=1021.315,104.835,-110.700,167.491,50.675,159.376
C07848=1021.309,104.587,-110.682,167.488,50.680,159.377
C07849=1021.303,104.337,-110.663,167.486,50.686,159.377
C07850=1021.297,104.088,-110.645,167.483,50.692,159.378
C07851=1021.292,103.838,-110.626,167.480,50.698,159.379
C07852=1021.287,103.590,-110.607,167.478,50.704,159.380
C07853=1021.281,103.340,-110.589,167.475,50.710,159.380
C07854=1021.276,103.091,-110.571,167.472,50.716,159.381
C07855=1021.270,102.841,-110.553,167.469,50.722,159.382
C07856=1021.265,102.593,-110.534,167.467,50.728,159.382
C07857=1021.259,102.343,-110.515,167.464,50.734,159.383
C07858=1021.253,102.094,-110.497,167.461,50.740,159.384
C07859=1021.248,101.844,-110.478,167.458,50.746,159.384
C07860=1021.242,101.595,-110.461,167.455,50.751,159.385
C07861=1021.237,101.346,-110.442,167.453,50.758,159.386
C07862=1021.232,101.096,-110.423,167.450,50.764,159.386
C07863=1021.226,100.848,-110.405,167.447,50.770,159.387
C07864=1021.221,100.598,-110.387,167.445,50.775,159.388
C07865=1021.215,100.349,-110.368,167.442,50.781,159.388
C07866=1021.210,100.099,-110.350,167.439,50.787,159.389
C07867=1021.204,99.850,-110.332,167.437,50.794,159.390
C07868=1021.198,99.601,-110.313,167.434,50.799,159.391
C07869=1021.194,99.351,-110.295,167.431,50.805,159.391
C07870=1021.188,99.102,-110.277,167.428,50.811,159.392
C07871=1021.182,98.853,-110.259,167.426,50.818,159.393
C07872=1021.177,98.604,-110.240,167.423,50.823,159.393
C07873=1021.171,98.354,-110.223,167.420,50.829,159.394
C07874=1021.165,98.105,-110.205,167.416,50.835,159.395
C07875=1021.160,97.856,-110.186,167.414,50.842,159.395
C07876=1021.154,97.607,-110.168,167.411,50.848,159.396
C07877=1021.149,97.358,-110.151,167.408,50.854,159.397
C07878=1021.142,97.108,-110.133,167.406,50.860,159.398
C07879=1021.137,96.859,-110.114,167.403,50.866,159.398
C07880=1021.131,96.609,-110.096,167.400,50.872,159.399
C07881=1021.126,96.360,-110.078,167.397,50.878,159.400
C07882=1021.121,96.111,-110.060,167.395,50.884,159.400
C07883=1021.115,95.861,-110.042,167.392,50.890,159.401
C07884=1021.109,95.613,-110.024,167.389,50.896,159.402
C07885=1021.104,95.363,-110.005,167.387,50.902,159.402
C07886=1021.098,95.114,-109.988,167.384,50.908,159.403
C07887=1021.093,94.865,-109.970,167.381,50.914,159.404
C07888=1021.086,94.615,-109.952,167.379,50.920,159.405
C07889=1021.082,94.366,-109.934,167.376,50.926,159.405
C07890=1021.076,94.117,-109.916,167.374,50.932,159.406
C07891=1021.070,93.868,-109.898,167.371,50.938,159.407
C07892=1021.065,93.618,-109.880,167.368,50.944,159.407
C07893=1021.059,93.369,-109.862,167.365,50.950,159.408
C07894=1021.053,93.119,-109.844,167.363,50.956,159.409
C07895=1021.048,92.870,-109.827,167.360,50.962,159.410
C07896=1021.043,92.621,-109.809,167.357,50.968,159.410
C07897=1021.037,92.371,-109.791,167.354,50.974,159.411
C07898=1021.031,92.122,-109.773,167.352,50.980,159.411
C07899=1021.026,91.873,-109.754,167.349,50.986,159.412
C07900=1021.019,91.590,-109.735,167.346,50.993,159.413
C07901=1021.013,91.307,-109.714,167.342,51.000,159.414
C07902=1021.007,91.023,-109.694,167.340,51.006,159.415
C07903=1021.001,90.741,-109.673,167.337,51.013,159.415
C07904=1020.995,90.491,-109.655,167.334,51.019,159.416
C07905=1020.990,90.242,-109.637,167.331,51.025,159.417
C07906=1020.984,89.993,-109.620,167.328,51.031,159.417
C07907=1020.979,89.744,-109.602,167.325,51.037,159.418
C07908=1020.974,89.494,-109.583,167.323,51.043,159.419
C07909=1020.968,89.245,-109.566,167.320,51.049,159.420
C07910=1020.963,88.996,-109.548,167.318,51.055,159.420
C07911=1020.956,88.746,-109.530,167.315,51.061,159.421
C07912=1020.951,88.497,-109.513,167.312,51.067,159.421
C07913=1020.946,88.247,-109.496,167.310,51.073,159.422
C07914=1020.940,87.997,-109.478,167.307,51.079,159.423
C07915=1020.934,87.748,-109.460,167.304,51.085,159.424
C07916=1020.929,87.499,-109.443,167.302,51.092,159.424
C07917=1020.923,87.250,-109.425,167.299,51.097,159.425
C07918=1020.917,87.001,-109.407,167.296,51.103,159.426
C07919=1020.911,86.751,-109.390,167.294,51.110,159.427
C07920=1020.906,86.502,-109.373,167.291,51.116,159.427
C07921=1020.901,86.253,-109.355,167.288,51.122,159.428
C07922=1020.895,86.003,-109.337,167.285,51.127,159.429
C07923=1020.889,85.754,-109.320,167.282,51.134,159.429
C07924=1020.883,85.505,-109.302,167.279,51.140,159.430
C07925=1020.878,85.255,-109.286,167.277,51.146,159.431
C07926=1020.872,85.006,-109.268,167.274,51.152,159.431
C07927=1020.867,84.757,-109.250,167.271,51.158,159.432
C07928=1020.861,84.507,-109.232,167.269,51.164,159.433
C07929=1020.856,84.258,-109.215,167.266,51.170,159.433
C07930=1020.849,84.008,-109.198,167.263,51.176,159.434
C07931=1020.844,83.759,-109.181,167.261,51.183,159.435
C07932=1020.838,83.510,-109.163,167.258,51.189,159.436
C07933=1020.832,83.261,-109.146,167.255,51.194,159.436
C07934=1020.827,83.012,-109.129,167.253,51.200,159.437
C07935=1020.821,82.762,-109.111,167.250,51.206,159.438
C07936=1020.816,82.513,-109.093,167.247,51.213,159.438
C07937=1020.810,82.264,-109.076,167.245,51.219,159.439
C07938=1020.805,82.014,-109.059,167.242,51.224,159.440
C07939=1020.799,81.765,-109.041,167.239,51.230,159.440
C07940=1020.794,81.516,-109.024,167.236,51.236,159.441
C07941=1020.788,81.266,-109.006,167.234,51.243,159.442
C07942=1020.783,81.017,-108.989,167.231,51.249,159.443
C07943=1020.777,80.768,-108.971,167.229,51.255,159.443
C07944=1020.772,80.518,-108.954,167.226,51.260,159.444
C07945=1020.766,80.269,-108.937,167.223,51.266,159.444
C07946=1020.761,80.020,-108.919,167.221,51.272,159.445
C07947=1020.755,79.770,-108.901,167.219,51.278,159.446
C07948=1020.749,79.520,-108.885,167.216,51.284,159.447
C07949=1020.744,79.271,-108.867,167.213,51.290,159.447
C07950=1020.739,79.022,-108.850,167.211,51.296,159.448
C07951=1020.733,78.773,-108.833,167.208,51.302,159.449
C07952=1020.728,78.524,-108.815,167.205,51.308,159.449
C07953=1020.722,78.274,-108.798,167.202,51.314,159.450
C07954=1020.717,78.025,-108.781,167.200,51.320,159.451
C07955=1020.711,77.775,-108.763,167.197,51.326,159.451
C07956=1020.706,77.526,-108.746,167.195,51.332,159.452
C07957=1020.699,77.277,-108.729,167.192,51.338,159.453
C07958=1020.694,77.027,-108.712,167.189,51.344,159.453
C07959=1020.689,76.778,-108.694,167.186,51.350,159.454
C07960=1020.683,76.528,-108.678,167.184,51.356,159.455
C07961=1020.678,76.279,-108.660,167.181,51.362,159.456
C07962=1020.672,76.030,-108.644,167.179,51.368,159.456
C07963=1020.666,75.781,-108.626,167.176,51.374,159.457
C07964=1020.660,75.498,-108.607,167.173,51.381,159.458
C07965=1020.653,75.215,-108.588,167.170,51.388,159.458
C07966=1020.647,74.931,-108.568,167.167,51.395,159.459
C07967=1020.641,74.648,-108.549,167.164,51.402,159.460
C07968=1020.635,74.399,-108.532,167.161,51.407,159.461
C07969=1020.630,74.150,-108.515,167.158,51.414,159.461
C07970=1020.624,73.900,-108.498,167.156,51.420,159.462
C07971=1020.618,73.651,-108.481,167.153,51.426,159.463
C07972=1020.612,73.401,-108.464,167.150,51.432,159.463
C07973=1020.607,73.152,-108.447,167.148,51.438,159.464
C07974=1020.601,72.902,-108.430,167.145,51.444,159.465
C07975=1020.596,72.653,-108.413,167.142,51.450,159.466
C07976=1020.590,72.404,-108.396,167.140,51.456,159.466
C07977=1020.584,72.154,-108.380,167.137,51.462,159.467
C07978=1020.579,71.905,-108.362,167.134,51.468,159.468
C07979=1020.573,71.656,-108.345,167.132,51.474,159.468
C07980=1020.568,71.406,-108.329,167.129,51.480,159.469
C07981=1020.562,71.157,-108.311,167.127,51.486,159.470
C07982=1020.557,70.908,-108.294,167.124,51.492,159.470
C07983=1020.551,70.658,-108.278,167.121,51.498,159.471
C07984=1020.546,70.409,-108.261,167.118,51.504,159.472
C07985=1020.539,70.160,-108.244,167.116,51.510,159.472
C07986=1020.534,69.910,-108.228,167.114,51.516,159.473
C07987=1020.529,69.661,-108.211,167.112,51.522,159.474
C07988=1020.523,69.412,-108.194,167.109,51.528,159.475
C07989=1020.517,69.162,-108.177,167.106,51.534,159.475
C07990=1020.512,68.913,-108.160,167.104,51.540,159.476
C07991=1020.506,68.663,-108.144,167.101,51.546,159.476
C07992=1020.501,68.414,-108.126,167.098,51.552,159.477
C07993=1020.495,68.165,-108.110,167.095,51.558,159.478
C07994=1020.490,67.915,-108.093,167.093,51.564,159.479
C07995=1020.484,67.666,-108.077,167.090,51.570,159.479
C07996=1020.478,67.416,-108.060,167.088,51.576,159.480
C07997=1020.472,67.167,-108.043,167.085,51.582,159.481
C07998=1020.467,66.918,-108.026,167.082,51.588,159.481
C07999=1020.461,66.668,-108.010,167.080,51.594,159.482
C08000=1020.456,66.419,-107.993,167.077,51.601,159.483
C08001=1020.450,66.169,-107.977,167.075,51.606,159.483
C08002=1020.445,65.920,-107.960,167.072,51.612,159.484
C08003=1020.439,65.670,-107.944,167.069,51.618,159.485
C08004=1020.433,65.421,-107.926,167.066,51.624,159.485
C08005=1020.427,65.172,-107.910,167.064,51.630,159.486
C08006=1020.421,64.923,-107.894,167.061,51.637,159.487
C08007=1020.416,64.673,-107.877,167.059,51.643,159.487
C08008=1020.410,64.424,-107.861,167.056,51.649,159.488
C08009=1020.406,64.175,-107.844,167.053,51.655,159.489
C08010=1020.400,63.925,-107.828,167.051,51.661,159.489
C08011=1020.394,63.676,-107.811,167.048,51.666,159.490
C08012=1020.388,63.426,-107.795,167.045,51.672,159.491
C08013=1020.382,63.177,-107.778,167.043,51.678,159.491
C08014=1020.377,62.927,-107.762,167.040,51.685,159.492
C08015=1020.371,62.678,-107.745,167.038,51.691,159.493
C08016=1020.365,62.429,-107.729,167.035,51.697,159.494
C08017=1020.359,62.179,-107.713,167.033,51.703,159.494
C08018=1020.353,61.930,-107.697,167.030,51.709,159.495
C08019=1020.348,61.680,-107.680,167.027,51.715,159.496
C08020=1020.343,61.430,-107.664,167.025,51.721,159.496
C08021=1020.337,61.181,-107.648,167.022,51.728,159.497
C08022=1020.331,60.932,-107.632,167.019,51.734,159.498
C08023=1020.325,60.682,-107.615,167.016,51.740,159.498
C08024=1020.319,60.434,-107.599,167.013,51.746,159.499
C08025=1020.313,60.184,-107.583,167.011,51.753,159.500
C08026=1020.307,59.935,-107.567,167.008,51.759,159.501
C08027=1020.303,59.685,-107.551,167.005,51.765,159.501
C08028=1020.296,59.402,-107.532,167.003,51.771,159.502
C08029=1020.289,59.118,-107.514,167.000,51.778,159.503
C08030=1020.282,58.835,-107.495,166.997,51.785,159.503
C08031=1020.276,58.552,-107.477,166.993,51.792,159.504
C08032=1020.270,58.302,-107.461,166.991,51.799,159.505
C08033=1020.264,58.053,-107.445,166.988,51.805,159.506
C08034=1020.259,57.803,-107.429,166.986,51.811,159.506
C08035=1020.253,57.555,-107.413,166.983,51.817,159.507
C08036=1020.247,57.305,-107.397,166.980,51.823,159.508
C08037=1020.241,57.056,-107.381,166.978,51.829,159.509
C08038=1020.236,56.806,-107.365,166.975,51.835,159.509
C08039=1020.231,56.556,-107.348,166.973,51.841,159.510
C08040=1020.225,56.307,-107.332,166.970,51.847,159.510
C08041=1020.219,56.058,-107.316,166.967,51.853,159.511
C08042=1020.214,55.808,-107.301,166.965,51.859,159.512
C08043=1020.208,55.559,-107.284,166.962,51.866,159.513
C08044=1020.202,55.310,-107.268,166.960,51.872,159.513
C08045=1020.196,55.060,-107.252,166.957,51.878,159.514
C08046=1020.191,54.811,-107.237,166.954,51.884,159.515
C08047=1020.185,54.562,-107.220,166.952,51.890,159.515
C08048=1020.179,54.312,-107.204,166.949,51.896,159.516
C08049=1020.174,54.063,-107.187,166.946,51.902,159.516
C08050=1020.168,53.813,-107.172,166.944,51.908,159.517
C08051=1020.163,53.564,-107.156,166.941,51.914,159.518
C08052=1020.157,53.315,-107.140,166.939,51.920,159.519
C08053=1020.151,53.065,-107.124,166.936,51.926,159.519
C08054=1020.145,52.815,-107.108,166.933,51.932,159.520
C08055=1020.139,52.566,-107.092,166.931,51.938,159.521
C08056=1020.134,52.317,-107.076,166.928,51.944,159.521
C08057=1020.128,52.067,-107.060,166.926,51.950,159.522
C08058=1020.122,51.818,-107.044,166.923,51.956,159.523
C08059=1020.117,51.568,-107.028,166.920,51.962,159.523
C08060=1020.112,51.319,-107.012,166.918,51.968,159.524
C08061=1020.106,51.069,-106.996,166.915,51.974,159.524
C08062=1020.100,50.820,-106.980,166.912,51.980,159.525
C08063=1020.095,50.571,-106.964,166.910,51.986,159.526
C08064=1020.089,50.321,-106.949,166.908,51.992,159.527
C08065=1020.083,50.072,-106.932,166.905,51.998,159.527
C08066=1020.077,49.822,-106.916,166.903,52.004,159.528
C08067=1020.072,49.573,-106.901,166.900,52.010,159.528
C08068=1020.066,49.324,-106.885,166.897,52.015,159.529
C08069=1020.061,49.074,-106.869,166.895,52.021,159.530
C08070=1020.056,48.825,-106.853,166.892,52.027,159.530
C08071=1020.051,48.575,-106.837,166.889,52.033,159.531
C08072=1020.045,48.326,-106.821,166.887,52.039,159.532
C08073=1020.039,48.076,-106.805,166.884,52.045,159.532
C08074=1020.034,47.827,-106.789,166.881,52.051,159.533
C08075=1020.028,47.578,-106.773,166.879,52.057,159.534
C08076=1020.022,47.328,-106.758,166.876,52.063,159.534
C08077=1020.017,47.079,-106.742,166.873,52.069,159.535
C08078=1020.011,46.829,-106.726,166.871,52.075,159.536
C08079=1020.005,46.580,-106.710,166.869,52.081,159.536
C08080=1020.000,46.330,-106.695,166.867,52.087,159.537
C08081=1019.994,46.081,-106.679,166.863,52.092,159.537
C08082=1019.989,45.831,-106.662,166.861,52.098,159.538
C08083=1019.984,45.582,-106.647,166.858,52.104,159.539
C08084=1019.978,45.332,-106.631,166.856,52.110,159.539
C08085=1019.973,45.084,-106.615,166.853,52.116,159.540
C08086=1019.967,44.834,-106.600,166.850,52.122,159.541
C08087=1019.961,44.584,-106.583,166.848,52.128,159.541
C08088=1019.956,44.335,-106.568,166.845,52.134,159.542
C08089=1019.950,44.086,-106.552,166.842,52.140,159.543
C08090=1019.945,43.836,-106.536,166.840,52.145,159.543
C08091=1019.939,43.587,-106.520,166.838,52.151,159.544
C08092=1019.934,43.303,-106.503,166.834,52.158,159.545
C08093=1019.927,43.020,-106.485,166.832,52.164,159.545
C08094=1019.921,42.736,-106.467,166.829,52.171,159.546
C08095=1019.914,42.453,-106.449,166.826,52.178,159.547
C08096=1019.909,42.203,-106.434,166.824,52.184,159.547
C08097=1019.903,41.954,-106.418,166.821,52.190,159.548
C08098=1019.898,41.704,-106.402,166.818,52.196,159.549
C08099=1019.892,41.454,-106.387,166.816,52.202,159.549
C08100=1019.886,41.206,-106.371,166.813,52.208,159.550
C08101=1019.880,40.956,-106.356,166.811,52.214,159.551
C08102=1019.875,40.707,-106.341,166.808,52.220,159.551
C08103=1019.870,40.457,-106.325,166.805,52.226,159.552
C08104=1019.863,40.208,-106.310,166.803,52.232,159.553
C08105=1019.858,39.959,-106.294,166.800,52.237,159.553
C08106=1019.852,39.709,-106.279,166.797,52.243,159.554
C08107=1019.847,39.459,-106.264,166.794,52.249,159.554
C08108=1019.842,39.209,-106.248,166.792,52.255,159.555
C08109=1019.836,38.961,-106.233,166.789,52.261,159.556
C08110=1019.830,38.711,-106.217,166.786,52.267,159.556
C08111=1019.825,38.462,-106.202,166.784,52.273,159.557
C08112=1019.819,38.212,-106.187,166.781,52.279,159.557
C08113=1019.813,37.963,-106.170,166.779,52.285,159.558
C08114=1019.807,37.714,-106.156,166.776,52.291,159.559
C08115=1019.802,37.464,-106.140,166.773,52.297,159.559
C08116=1019.797,37.214,-106.125,166.771,52.303,159.560
C08117=1019.791,36.964,-106.110,166.768,52.309,159.560
C08118=1019.785,36.715,-106.095,166.766,52.314,159.561
C08119=1019.780,36.465,-106.079,166.764,52.320,159.562
C08120=1019.775,36.216,-106.064,166.761,52.326,159.563
C08121=1019.768,35.967,-106.049,166.758,52.332,159.563
C08122=1019.763,35.717,-106.034,166.756,52.338,159.564
C08123=1019.757,35.468,-106.019,166.752,52.345,159.564
C08124=1019.751,35.218,-106.004,166.749,52.351,159.565
C08125=1019.745,34.969,-105.989,166.747,52.357,159.566
C08126=1019.740,34.719,-105.973,166.744,52.363,159.566
C08127=1019.734,34.470,-105.959,166.742,52.369,159.567
C08128=1019.728,34.220,-105.943,166.739,52.375,159.568
C08129=1019.723,33.971,-105.928,166.736,52.381,159.568
C08130=1019.717,33.721,-105.913,166.734,52.387,159.569
C08131=1019.712,33.472,-105.898,166.731,52.393,159.570
C08132=1019.706,33.223,-105.883,166.730,52.399,159.570
C08133=1019.700,32.973,-105.868,166.727,52.405,159.571
C08134=1019.695,32.724,-105.853,166.724,52.411,159.572
C08135=1019.689,32.474,-105.838,166.722,52.417,159.572
C08136=1019.683,32.225,-105.823,166.719,52.423,159.573
C08137=1019.678,31.975,-105.808,166.717,52.429,159.574
C08138=1019.672,31.726,-105.793,166.714,52.435,159.574
C08139=1019.666,31.476,-105.778,166.711,52.440,159.575
C08140=1019.660,31.227,-105.763,166.708,52.446,159.575
C08141=1019.655,30.977,-105.747,166.706,52.452,159.576
C08142=1019.649,30.728,-105.733,166.703,52.458,159.577
C08143=1019.644,30.479,-105.718,166.701,52.464,159.577
C08144=1019.638,30.229,-105.703,166.698,52.470,159.578
C08145=1019.633,29.979,-105.688,166.695,52.476,159.578
C08146=1019.627,29.729,-105.673,166.693,52.482,159.579
C08147=1019.621,29.480,-105.658,166.690,52.488,159.580
C08148=1019.616,29.230,-105.643,166.687,52.494,159.580
C08149=1019.610,28.981,-105.628,166.685,52.500,159.581
C08150=1019.605,28.732,-105.613,166.682,52.506,159.581
C08151=1019.599,28.482,-105.598,166.679,52.512,159.582
C08152=1019.594,28.233,-105.583,166.676,52.517,159.583
C08153=1019.587,27.983,-105.569,166.674,52.523,159.583
C08154=1019.582,27.734,-105.553,166.671,52.529,159.584
C08155=1019.577,27.485,-105.539,166.669,52.535,159.584
C08156=1019.570,27.201,-105.522,166.666,52.542,159.585
C08157=1019.564,26.917,-105.505,166.663,52.548,159.586
C08158=1019.557,26.634,-105.489,166.660,52.556,159.587
C08159=1019.551,26.351,-105.472,166.657,52.562,159.587
C08160=1019.545,26.101,-105.457,166.655,52.568,159.588
C08161=1019.540,25.852,-105.442,166.652,52.574,159.589
C08162=1019.534,25.601,-105.428,166.649,52.580,159.589
C08163=1019.528,25.352,-105.413,166.647,52.586,159.590
C08164=1019.523,25.103,-105.398,166.644,52.592,159.590
C08165=1019.517,24.853,-105.384,166.641,52.598,159.591
C08166=1019.511,24.604,-105.369,166.639,52.604,159.592
C08167=1019.505,24.355,-105.354,166.636,52.610,159.592
C08168=1019.500,24.104,-105.340,166.634,52.616,159.593
C08169=1019.494,23.855,-105.325,166.631,52.622,159.594
C08170=1019.488,23.606,-105.310,166.628,52.627,159.594
C08171=1019.482,23.356,-105.296,166.626,52.634,159.595
C08172=1019.477,23.107,-105.281,166.623,52.640,159.595
C08173=1019.472,22.857,-105.267,166.620,52.646,159.596
C08174=1019.465,22.608,-105.252,166.618,52.652,159.597
C08175=1019.460,22.358,-105.237,166.615,52.658,159.597
C08176=1019.455,22.109,-105.223,166.612,52.663,159.598
C08177=1019.448,21.859,-105.208,166.610,52.669,159.598
C08178=1019.443,21.610,-105.194,166.607,52.675,159.599
C08179=1019.438,21.360,-105.179,166.605,52.681,159.600
C08180=1019.432,21.111,-105.165,166.602,52.687,159.600
C08181=1019.426,20.861,-105.150,166.599,52.693,159.601
C08182=1019.420,20.612,-105.136,166.596,52.699,159.601
C08183=1019.415,20.362,-105.121,166.594,52.705,159.602
C08184=1019.409,20.113,-105.106,166.591,52.711,159.603
C08185=1019.404,19.863,-105.093,166.589,52.717,159.603
C08186=1019.399,19.614,-105.077,166.586,52.722,159.604
C08187=1019.393,19.364,-105.064,166.583,52.728,159.604
C08188=1019.387,19.115,-105.049,166.581,52.734,159.605
C08189=1019.381,18.865,-105.035,166.578,52.741,159.606
C08190=1019.375,18.616,-105.020,166.575,52.747,159.606
C08191=1019.370,18.366,-105.006,166.572,52.752,159.607
C08192=1019.365,18.116,-104.991,166.570,52.758,159.607
C08193=1019.359,17.867,-104.977,166.567,52.764,159.608
C08194=1019.353,17.617,-104.963,166.565,52.770,159.609
C08195=1019.348,17.368,-104.948,166.562,52.776,159.609
C08196=1019.342,17.118,-104.934,166.559,52.782,159.610
C08197=1019.336,16.869,-104.920,166.557,52.788,159.610
C08198=1019.330,16.620,-104.906,166.554,52.794,159.611
C08199=1019.325,16.370,-104.892,166.552,52.800,159.612
C08200=1019.319,16.121,-104.877,166.549,52.806,159.612
C08201=1019.314,15.870,-104.862,166.546,52.811,159.613
C08202=1019.308,15.621,-104.849,166.543,52.817,159.613
C08203=1019.302,15.372,-104.834,166.541,52.823,159.614
C08204=1019.297,15.122,-104.820,166.538,52.830,159.615
C08205=1019.291,14.873,-104.806,166.535,52.835,159.615
C08206=1019.285,14.623,-104.791,166.533,52.841,159.616
C08207=1019.280,14.374,-104.778,166.530,52.847,159.616
C08208=1019.274,14.124,-104.764,166.528,52.853,159.617
C08209=1019.268,13.875,-104.749,166.525,52.859,159.617
C08210=1019.264,13.625,-104.735,166.522,52.865,159.618
C08211=1019.258,13.375,-104.720,166.520,52.871,159.619
C08212=1019.252,13.125,-104.707,166.517,52.877,159.619
C08213=1019.246,12.877,-104.693,166.515,52.883,159.620
C08214=1019.240,12.627,-104.679,166.512,52.889,159.620
C08215=1019.235,12.377,-104.665,166.509,52.894,159.621
C08216=1019.229,12.128,-104.651,166.506,52.900,159.622
C08217=1019.223,11.878,-104.637,166.504,52.907,159.622
C08218=1019.218,11.628,-104.623,166.500,52.913,159.623
C08219=1019.211,11.379,-104.609,166.498,52.919,159.623
C08220=1019.205,11.097,-104.593,166.496,52.926,159.624
C08221=1019.199,10.816,-104.578,166.492,52.932,159.625
C08222=1019.192,10.533,-104.562,166.489,52.939,159.625
C08223=1019.186,10.251,-104.546,166.485,52.946,159.626
C08224=1019.180,10.002,-104.533,166.483,52.952,159.627
C08225=1019.174,9.753,-104.519,166.480,52.958,159.627
C08226=1019.169,9.503,-104.505,166.478,52.964,159.628
C08227=1019.163,9.253,-104.491,166.475,52.970,159.628
C08228=1019.157,9.003,-104.477,166.473,52.976,159.629
C08229=1019.152,8.754,-104.463,166.470,52.982,159.630
C08230=1019.145,8.504,-104.450,166.467,52.988,159.630
C08231=1019.140,8.255,-104.436,166.465,52.994,159.631
C08232=1019.134,8.005,-104.422,166.462,53.000,159.631
C08233=1019.129,7.756,-104.408,166.460,53.006,159.632
C08234=1019.124,7.506,-104.394,166.457,53.012,159.633
C08235=1019.117,7.257,-104.381,166.454,53.018,159.633
C08236=1019.112,7.007,-104.367,166.452,53.024,159.634
C08237=1019.106,6.758,-104.353,166.449,53.030,159.634
C08238=1019.101,6.508,-104.339,166.445,53.036,159.635
C08239=1019.095,6.258,-104.325,166.442,53.042,159.635
C08240=1019.089,6.009,-104.312,166.440,53.048,159.636
C08241=1019.083,5.759,-104.298,166.437,53.054,159.637
C08242=1019.078,5.509,-104.284,166.434,53.059,159.637
C08243=1019.072,5.260,-104.270,166.432,53.066,159.638
C08244=1019.067,5.010,-104.256,166.429,53.072,159.638
C08245=1019.061,4.761,-104.243,166.427,53.078,159.639
C08246=1019.055,4.511,-104.229,166.424,53.083,159.639
C08247=1019.050,4.262,-104.215,166.421,53.089,159.640
C08248=1019.044,4.012,-104.202,166.419,53.095,159.641
C08249=1019.039,3.763,-104.188,166.416,53.101,159.641
C08250=1019.033,3.513,-104.174,166.413,53.107,159.642
C08251=1019.027,3.264,-104.161,166.411,53.113,159.642
C08252=1019.021,3.014,-104.147,166.408,53.119,159.643
C08253=1019.016,2.765,-104.133,166.405,53.125,159.643
C08254=1019.010,2.515,-104.119,166.403,53.131,159.644
C08255=1019.005,2.265,-104.105,166.400,53.137,159.645
C08256=1018.999,2.016,-104.093,166.397,53.142,159.645
C08257=1018.994,1.766,-104.079,166.395,53.148,159.646
C08258=1018.988,1.516,-104.065,166.392,53.154,159.646
C08259=1018.983,1.267,-104.051,166.389,53.160,159.647
C08260=1018.977,1.017,-104.037,166.387,53.166,159.647
C08261=1018.972,0.769,-104.024,166.384,53.171,159.648
C08262=1018.966,0.519,-104.010,166.381,53.177,159.648
C08263=1018.961,0.269,-103.997,166.379,53.184,159.649
C08264=1018.955,0.019,-103.983,166.376,53.189,159.650
C08265=1018.949,-0.230,-103.970,166.373,53.195,159.650
C08266=1018.944,-0.479,-103.956,166.371,53.201,159.651
C08267=1018.938,-0.729,-103.942,166.368,53.207,159.651
C08268=1018.933,-0.979,-103.928,166.365,53.213,159.652
C08269=1018.928,-1.229,-103.915,166.363,53.218,159.652
C08270=1018.921,-1.478,-103.902,166.360,53.224,159.653
C08271=1018.916,-1.728,-103.888,166.357,53.230,159.653
C08272=1018.910,-1.977,-103.874,166.355,53.236,159.654
C08273=1018.905,-2.227,-103.860,166.352,53.241,159.654
C08274=1018.900,-2.476,-103.848,166.349,53.247,159.655
C08275=1018.894,-2.726,-103.834,166.346,53.253,159.655
C08276=1018.889,-2.975,-103.820,166.344,53.259,159.656
C08277=1018.883,-3.225,-103.807,166.341,53.265,159.657
C08278=1018.878,-3.475,-103.793,166.338,53.271,159.657
C08279=1018.872,-3.724,-103.780,166.336,53.277,159.658
C08280=1018.866,-3.974,-103.766,166.333,53.282,159.658
C08281=1018.861,-4.224,-103.753,166.330,53.288,159.659
C08282=1018.856,-4.473,-103.739,166.327,53.294,159.659
C08283=1018.850,-4.723,-103.726,166.325,53.300,159.660
C08284=1018.844,-5.003,-103.712,166.321,53.306,159.660
C08285=1018.837,-5.283,-103.697,166.318,53.313,159.661
C08286=1018.831,-5.563,-103.683,166.315,53.320,159.662
C08287=1018.825,-5.842,-103.668,166.313,53.327,159.662
C08288=1018.819,-6.092,-103.655,166.309,53.333,159.663
C08289=1018.813,-6.342,-103.641,166.306,53.339,159.663
C08290=1018.808,-6.592,-103.629,166.304,53.345,159.664
C08291=1018.802,-6.841,-103.615,166.301,53.351,159.665
C08292=1018.796,-7.091,-103.602,166.298,53.357,159.665
C08293=1018.790,-7.340,-103.589,166.296,53.363,159.666
C08294=1018.785,-7.590,-103.576,166.293,53.369,159.666
C08295=1018.779,-7.839,-103.563,166.290,53.374,159.667
C08296=1018.774,-8.089,-103.550,166.288,53.380,159.667
C08297=1018.768,-8.338,-103.536,166.284,53.387,159.668
C08298=1018.762,-8.588,-103.524,166.281,53.392,159.668
C08299=1018.757,-8.838,-103.511,166.279,53.398,159.669
C08300=1018.751,-9.087,-103.498,166.276,53.405,159.670
C08301=1018.746,-9.337,-103.485,166.273,53.410,159.670
C08302=1018.740,-9.587,-103.471,166.271,53.416,159.671
C08303=1018.735,-9.837,-103.458,166.269,53.422,159.671
C08304=1018.729,-10.085,-103.445,166.266,53.428,159.672
C08305=1018.723,-10.335,-103.433,166.263,53.434,159.672
C08306=1018.718,-10.585,-103.420,166.261,53.440,159.673
C08307=1018.712,-10.835,-103.406,166.257,53.446,159.673
C08308=1018.707,-11.084,-103.394,166.254,53.452,159.674
C08309=1018.701,-11.333,-103.380,166.251,53.458,159.674
C08310=1018.695,-11.583,-103.368,166.249,53.464,159.675
C08311=1018.690,-11.834,-103.355,166.246,53.470,159.675
C08312=1018.684,-12.082,-103.342,166.243,53.475,159.676
C08313=1018.679,-12.332,-103.329,166.241,53.481,159.677
C08314=1018.673,-12.582,-103.316,166.238,53.487,159.677
C08315=1018.667,-12.831,-103.303,166.235,53.493,159.678
C08316=1018.662,-13.081,-103.290,166.233,53.499,159.678
C08317=1018.656,-13.331,-103.277,166.230,53.505,159.679
C08318=1018.651,-13.580,-103.264,166.227,53.511,159.679
C08319=1018.646,-13.830,-103.251,166.224,53.517,159.679
C08320=1018.640,-14.079,-103.239,166.221,53.523,159.680
C08321=1018.635,-14.330,-103.226,166.218,53.528,159.681
C08322=1018.629,-14.578,-103.213,166.216,53.534,159.681
C08323=1018.624,-14.828,-103.200,166.213,53.540,159.682
C08324=1018.618,-15.078,-103.187,166.210,53.546,159.682
C08325=1018.612,-15.327,-103.174,166.207,53.551,159.683
C08326=1018.607,-15.577,-103.161,166.205,53.558,159.683
C08327=1018.601,-15.827,-103.148,166.202,53.563,159.684
C08328=1018.596,-16.076,-103.136,166.200,53.569,159.684
C08329=1018.591,-16.326,-103.123,166.197,53.575,159.685
C08330=1018.585,-16.576,-103.111,166.193,53.581,159.685
C08331=1018.579,-16.825,-103.098,166.191,53.587,159.686
C08332=1018.573,-17.075,-103.085,166.188,53.594,159.686
C08333=1018.567,-17.324,-103.073,166.185,53.599,159.687
C08334=1018.562,-17.574,-103.060,166.183,53.605,159.688
C08335=1018.556,-17.824,-103.048,166.180,53.611,159.688
C08336=1018.550,-18.073,-103.035,166.176,53.617,159.688
C08337=1018.546,-18.323,-103.022,166.174,53.623,159.689
C08338=1018.540,-18.573,-103.010,166.172,53.630,159.690
C08339=1018.534,-18.823,-102.997,166.169,53.635,159.690
C08340=1018.529,-19.072,-102.985,166.166,53.641,159.691
C08341=1018.523,-19.322,-102.973,166.163,53.647,159.691
C08342=1018.517,-19.571,-102.960,166.160,53.653,159.692
C08343=1018.511,-19.821,-102.948,166.157,53.659,159.692
C08344=1018.505,-20.071,-102.935,166.154,53.665,159.693
C08345=1018.500,-20.320,-102.923,166.152,53.671,159.693
C08346=1018.495,-20.570,-102.910,166.149,53.677,159.694
C08347=1018.490,-20.819,-102.898,166.147,53.683,159.694
C08348=1018.480,-21.237,-102.877,166.141,53.693,159.695
C08349=1018.471,-21.656,-102.856,166.137,53.703,159.696
C08350=1018.462,-22.074,-102.835,166.132,53.713,159.697
C08351=1018.452,-22.493,-102.815,166.127,53.722,159.698
C08352=1018.446,-22.743,-102.802,166.125,53.729,159.698
C08353=1018.441,-22.992,-102.790,166.122,53.734,159.699
C08354=1018.435,-23.242,-102.777,166.119,53.740,159.699
C08355=1018.430,-23.491,-102.765,166.116,53.746,159.700
C08356=1018.425,-23.741,-102.752,166.114,53.752,159.700
C08357=1018.419,-23.990,-102.740,166.110,53.758,159.701
C08358=1018.413,-24.240,-102.727,166.108,53.764,159.701
C08359=1018.408,-24.489,-102.715,166.105,53.770,159.702
C08360=1018.402,-24.739,-102.703,166.102,53.776,159.702
C08361=1018.397,-24.988,-102.690,166.099,53.781,159.703
C08362=1018.391,-25.239,-102.679,166.097,53.787,159.703
C08363=1018.386,-25.488,-102.666,166.094,53.793,159.704
C08364=1018.378,-25.847,-102.649,166.089,53.802,159.704
C08365=1018.370,-26.206,-102.630,166.086,53.810,159.705
C08366=1018.362,-26.565,-102.612,166.082,53.818,159.706
C08367=1018.354,-26.925,-102.595,166.078,53.827,159.707
C08368=1018.349,-27.174,-102.583,166.075,53.833,159.707
C08369=1018.343,-27.424,-102.570,166.072,53.839,159.708
C08370=1018.338,-27.673,-102.558,166.069,53.844,159.708
C08371=1018.332,-27.924,-102.546,166.067,53.851,159.709
C08372=1018.327,-28.173,-102.534,166.064,53.856,159.709
C08373=1018.322,-28.422,-102.522,166.061,53.863,159.709
C08374=1018.315,-28.672,-102.511,166.058,53.869,159.710
C08375=1018.310,-28.922,-102.498,166.055,53.874,159.711
C08376=1018.304,-29.172,-102.486,166.053,53.881,159.711
C08377=1018.299,-29.421,-102.474,166.049,53.886,159.711
C08378=1018.293,-29.671,-102.462,166.046,53.893,159.712
C08379=1018.287,-29.921,-102.451,166.044,53.899,159.713
C08380=1018.282,-30.170,-102.439,166.041,53.904,159.713
C08381=1018.276,-30.420,-102.426,166.039,53.911,159.714
C08382=1018.271,-30.670,-102.415,166.035,53.916,159.714
C08383=1018.265,-30.919,-102.402,166.032,53.923,159.715
C08384=1018.260,-31.169,-102.391,166.030,53.928,159.715
C08385=1018.254,-31.418,-102.379,166.027,53.934,159.716
C08386=1018.248,-31.668,-102.367,166.024,53.940,159.716
C08387=1018.243,-31.918,-102.355,166.021,53.946,159.716
C08388=1018.238,-32.167,-102.343,166.018,53.952,159.717
C08389=1018.232,-32.417,-102.331,166.015,53.958,159.718
C08390=1018.226,-32.666,-102.319,166.013,53.964,159.718
C08391=1018.221,-32.917,-102.308,166.010,53.970,159.719
C08392=1018.215,-33.166,-102.295,166.007,53.976,159.719
C08393=1018.210,-33.416,-102.284,166.004,53.982,159.719
C08394=1018.205,-33.666,-102.271,166.001,53.988,159.720
C08395=1018.199,-33.915,-102.261,165.999,53.994,159.720
C08396=1018.194,-34.164,-102.248,165.996,53.999,159.721
C08397=1018.188,-34.415,-102.236,165.993,54.005,159.721
C08398=1018.183,-34.664,-102.224,165.989,54.011,159.722
C08399=1018.178,-34.914,-102.213,165.987,54.018,159.722
C08400=1018.172,-35.163,-102.201,165.984,54.023,159.723
C08401=1018.166,-35.413,-102.189,165.982,54.029,159.723
C08402=1018.161,-35.662,-102.177,165.979,54.035,159.724
C08403=1018.156,-35.912,-102.166,165.975,54.041,159.724
C08404=1018.150,-36.162,-102.153,165.972,54.047,159.725
C08405=1018.144,-36.412,-102.142,165.970,54.053,159.725
C08406=1018.139,-36.661,-102.131,165.967,54.059,159.726
C08407=1018.134,-36.911,-102.119,165.964,54.064,159.726
C08408=1018.128,-37.188,-102.106,165.961,54.071,159.727
C08409=1018.122,-37.466,-102.092,165.957,54.077,159.727
C08410=1018.116,-37.743,-102.079,165.955,54.084,159.728
C08411=1018.109,-38.020,-102.066,165.951,54.090,159.728
C08412=1018.104,-38.270,-102.055,165.949,54.096,159.729
C08413=1018.099,-38.520,-102.043,165.946,54.102,159.729
C08414=1018.093,-38.769,-102.031,165.943,54.109,159.730
C08415=1018.088,-39.019,-102.020,165.940,54.114,159.730
C08416=1018.082,-39.269,-102.008,165.937,54.120,159.730
C08417=1018.077,-39.518,-101.996,165.935,54.126,159.731
C08418=1018.072,-39.768,-101.985,165.932,54.131,159.731
C08419=1018.066,-40.017,-101.974,165.928,54.138,159.732
C08420=1018.060,-40.268,-101.962,165.925,54.143,159.732
C08421=1018.055,-40.517,-101.951,165.923,54.150,159.733
C08422=1018.049,-40.767,-101.939,165.920,54.155,159.733
C08423=1018.044,-41.016,-101.928,165.917,54.162,159.734
C08424=1018.039,-41.266,-101.917,165.914,54.168,159.734
C08425=1018.032,-41.516,-101.905,165.912,54.174,159.735
C08426=1018.027,-41.766,-101.894,165.909,54.180,159.735
C08427=1018.021,-42.015,-101.883,165.905,54.186,159.736
C08428=1018.016,-42.265,-101.871,165.903,54.192,159.736
C08429=1018.010,-42.514,-101.860,165.900,54.198,159.737
C08430=1018.005,-42.765,-101.848,165.898,54.204,159.737
C08431=1017.999,-43.014,-101.837,165.894,54.210,159.738
C08432=1017.994,-43.264,-101.826,165.891,54.215,159.738
C08433=1017.988,-43.513,-101.815,165.888,54.221,159.739
C08434=1017.983,-43.763,-101.803,165.886,54.227,159.739
C08435=1017.978,-44.013,-101.792,165.882,54.234,159.739
C08436=1017.972,-44.262,-101.780,165.879,54.239,159.740
C08437=1017.966,-44.512,-101.769,165.877,54.245,159.741
C08438=1017.961,-44.762,-101.758,165.874,54.251,159.741
C08439=1017.955,-45.011,-101.747,165.871,54.258,159.741
C08440=1017.950,-45.261,-101.735,165.868,54.263,159.742
C08441=1017.944,-45.511,-101.724,165.865,54.269,159.742
C08442=1017.939,-45.760,-101.713,165.863,54.275,159.743
C08443=1017.934,-46.010,-101.702,165.860,54.280,159.743
C08444=1017.929,-46.260,-101.691,165.856,54.287,159.744
C08445=1017.923,-46.509,-101.680,165.853,54.293,159.744
C08446=1017.918,-46.759,-101.668,165.851,54.298,159.744
C08447=1017.912,-47.008,-101.657,165.848,54.304,159.745
C08448=1017.907,-47.259,-101.645,165.844,54.310,159.745
C08449=1017.901,-47.508,-101.635,165.842,54.317,159.746
C08450=1017.896,-47.758,-101.623,165.839,54.322,159.746
C08451=1017.890,-48.008,-101.612,165.836,54.328,159.747
C08452=1017.885,-48.258,-101.601,165.834,54.334,159.747
C08453=1017.879,-48.507,-101.590,165.830,54.340,159.748
C08454=1017.874,-48.757,-101.578,165.827,54.345,159.748
C08455=1017.869,-49.006,-101.568,165.825,54.352,159.749
C08456=1017.864,-49.256,-101.556,165.822,54.357,159.749
C08457=1017.858,-49.506,-101.545,165.819,54.363,159.749
C08458=1017.853,-49.755,-101.534,165.816,54.369,159.750
C08459=1017.847,-50.005,-101.523,165.813,54.375,159.750
C08460=1017.842,-50.255,-101.511,165.810,54.380,159.751
C08461=1017.836,-50.504,-101.500,165.808,54.387,159.751
C08462=1017.832,-50.755,-101.490,165.805,54.392,159.752
C08463=1017.826,-51.004,-101.479,165.802,54.398,159.752
C08464=1017.821,-51.254,-101.467,165.798,54.404,159.752
C08465=1017.815,-51.503,-101.457,165.796,54.410,159.753
C08466=1017.810,-51.753,-101.446,165.792,54.417,159.753
C08467=1017.804,-52.003,-101.435,165.790,54.423,159.754
C08468=1017.798,-52.252,-101.425,165.787,54.428,159.754
///RCONF 1,0,0,1,0,0,0,0,0,0,0,0,0,0,0,0,0,0,0,0,0,0,0,0
C08469=1017.793,-52.503,-101.414,165.784,54.435,159.755
C08470=1017.787,-52.752,-101.404,165.781,54.441,159.755
C08471=1017.781,-53.002,-101.393,165.778,54.447,159.756
C08472=1017.776,-53.279,-101.381,165.775,54.454,159.756
C08473=1017.770,-53.557,-101.369,165.772,54.460,159.757
C08474=1017.764,-53.834,-101.358,165.768,54.467,159.757
C08475=1017.757,-54.112,-101.345,165.765,54.474,159.758
C08476=1017.752,-54.362,-101.335,165.762,54.480,159.758
C08477=1017.746,-54.611,-101.324,165.759,54.487,159.759
C08478=1017.741,-54.861,-101.314,165.756,54.492,159.759
C08479=1017.735,-55.111,-101.303,165.754,54.498,159.760
C08480=1017.729,-55.360,-101.292,165.750,54.504,159.760
C08481=1017.724,-55.610,-101.282,165.748,54.511,159.761
C08482=1017.719,-55.859,-101.271,165.745,54.516,159.761
C08483=1017.713,-56.109,-101.261,165.741,54.523,159.762
C08484=1017.708,-56.359,-101.250,165.738,54.528,159.762
C08485=1017.703,-56.609,-101.240,165.736,54.535,159.763
C08486=1017.697,-56.859,-101.229,165.732,54.541,159.763
C08487=1017.692,-57.109,-101.219,165.730,54.547,159.763
C08488=1017.686,-57.358,-101.208,165.727,54.553,159.764
C08489=1017.680,-57.608,-101.197,165.723,54.558,159.764
C08490=1017.675,-57.857,-101.187,165.721,54.565,159.765
C08491=1017.670,-58.107,-101.176,165.718,54.570,159.765
C08492=1017.664,-58.357,-101.166,165.715,54.577,159.765
C08493=1017.658,-58.606,-101.155,165.712,54.583,159.766
C08494=1017.653,-58.856,-101.145,165.709,54.589,159.766
C08495=1017.647,-59.106,-101.134,165.706,54.595,159.767
C08496=1017.642,-59.356,-101.124,165.703,54.601,159.767
C08497=1017.638,-59.606,-101.113,165.700,54.607,159.768
C08498=1017.632,-59.855,-101.103,165.697,54.613,159.768
C08499=1017.627,-60.105,-101.092,165.694,54.619,159.769
C08500=1017.621,-60.355,-101.082,165.691,54.625,159.769
C08501=1017.615,-60.605,-101.071,165.689,54.631,159.770
C08502=1017.610,-60.854,-101.061,165.685,54.637,159.770
C08503=1017.605,-61.104,-101.051,165.682,54.642,159.770
C08504=1017.599,-61.354,-101.041,165.680,54.649,159.771
C08505=1017.594,-61.603,-101.030,165.676,54.655,159.771
C08506=1017.589,-61.853,-101.020,165.673,54.660,159.771
C08507=1017.583,-62.102,-101.009,165.671,54.666,159.772
C08508=1017.578,-62.352,-100.999,165.668,54.672,159.772
C08509=1017.572,-62.603,-100.989,165.664,54.678,159.773
C08510=1017.567,-62.851,-100.978,165.662,54.684,159.773
C08511=1017.562,-63.101,-100.968,165.659,54.690,159.774
C08512=1017.556,-63.352,-100.958,165.656,54.695,159.774
C08513=1017.551,-63.601,-100.946,165.653,54.702,159.774
C08514=1017.546,-63.851,-100.937,165.650,54.708,159.775
C08515=1017.541,-64.101,-100.926,165.647,54.713,159.775
C08516=1017.535,-64.350,-100.916,165.644,54.720,159.776
C08517=1017.530,-64.600,-100.905,165.641,54.726,159.776
C08518=1017.525,-64.850,-100.896,165.638,54.731,159.776
C08519=1017.519,-65.099,-100.885,165.636,54.737,159.777
C08520=1017.514,-65.349,-100.875,165.632,54.743,159.777
C08521=1017.509,-65.599,-100.865,165.629,54.749,159.778
C08522=1017.503,-65.848,-100.854,165.627,54.755,159.778
C08523=1017.498,-66.098,-100.844,165.624,54.761,159.779
C08524=1017.493,-66.348,-100.834,165.620,54.767,159.779
C08525=1017.487,-66.598,-100.824,165.618,54.773,159.779
C08526=1017.482,-66.847,-100.813,165.615,54.778,159.780
C08527=1017.477,-67.097,-100.803,165.612,54.784,159.780
C08528=1017.471,-67.347,-100.793,165.609,54.790,159.781
C08529=1017.466,-67.597,-100.783,165.606,54.796,159.781
C08530=1017.461,-67.846,-100.772,165.603,54.802,159.781
C08531=1017.455,-68.096,-100.762,165.600,54.807,159.782
C08532=1017.451,-68.345,-100.752,165.598,54.814,159.782
C08533=1017.445,-68.595,-100.742,165.594,54.819,159.782
C08534=1017.441,-68.846,-100.731,165.591,54.825,159.783
C08535=1017.435,-69.095,-100.721,165.588,54.831,159.783
C08536=1017.429,-69.373,-100.710,165.585,54.837,159.784
C08537=1017.423,-69.652,-100.699,165.582,54.844,159.784
C08538=1017.418,-69.931,-100.687,165.578,54.850,159.784
C08539=1017.412,-70.209,-100.676,165.575,54.856,159.785
C08540=1017.406,-70.459,-100.666,165.572,54.862,159.785
C08541=1017.401,-70.709,-100.656,165.569,54.869,159.786
C08542=1017.396,-70.959,-100.646,165.566,54.874,159.786
C08543=1017.390,-71.209,-100.636,165.564,54.880,159.787
C08544=1017.386,-71.458,-100.626,165.561,54.886,159.787
C08545=1017.380,-71.709,-100.616,165.557,54.892,159.787
C08546=1017.375,-71.958,-100.606,165.554,54.897,159.788
C08547=1017.370,-72.208,-100.596,165.551,54.903,159.788
C08548=1017.366,-72.457,-100.585,165.549,54.908,159.788
C08549=1017.360,-72.707,-100.575,165.546,54.914,159.789
C08550=1017.355,-72.957,-100.565,165.542,54.921,159.789
C08551=1017.350,-73.207,-100.555,165.540,54.926,159.790
C08552=1017.345,-73.456,-100.545,165.537,54.932,159.790
C08553=1017.340,-73.706,-100.535,165.534,54.937,159.790
C08554=1017.335,-73.956,-100.525,165.531,54.943,159.791
C08555=1017.329,-74.206,-100.515,165.528,54.949,159.791
C08556=1017.324,-74.455,-100.505,165.525,54.955,159.791
C08557=1017.319,-74.705,-100.495,165.522,54.960,159.792
C08558=1017.313,-74.954,-100.486,165.519,54.966,159.792
C08559=1017.308,-75.205,-100.475,165.517,54.972,159.793
C08560=1017.303,-75.455,-100.466,165.513,54.978,159.793
C08561=1017.297,-75.704,-100.457,165.510,54.984,159.793
C08562=1017.292,-75.954,-100.447,165.508,54.990,159.794
C08563=1017.287,-76.204,-100.437,165.504,54.996,159.794
C08564=1017.282,-76.453,-100.427,165.501,55.002,159.794
C08565=1017.276,-76.703,-100.417,165.498,55.007,159.795
C08566=1017.272,-76.953,-100.408,165.495,55.014,159.795
C08567=1017.266,-77.203,-100.398,165.492,55.020,159.796
C08568=1017.261,-77.452,-100.389,165.489,55.025,159.796
C08569=1017.256,-77.702,-100.379,165.487,55.031,159.796
C08570=1017.251,-77.952,-100.370,165.483,55.038,159.797
C08571=1017.246,-78.202,-100.360,165.481,55.043,159.797
C08572=1017.240,-78.452,-100.350,165.478,55.049,159.798
C08573=1017.235,-78.701,-100.341,165.475,55.055,159.798
C08574=1017.229,-78.951,-100.330,165.471,55.061,159.798
C08575=1017.224,-79.201,-100.322,165.469,55.067,159.799
C08576=1017.219,-79.450,-100.312,165.466,55.073,159.799
C08577=1017.214,-79.700,-100.302,165.462,55.079,159.799
C08578=1017.209,-79.950,-100.293,165.459,55.084,159.800
C08579=1017.204,-80.200,-100.284,165.457,55.090,159.800
C08580=1017.198,-80.450,-100.274,165.454,55.095,159.800
C08581=1017.193,-80.699,-100.265,165.451,55.102,159.801
C08582=1017.188,-80.949,-100.255,165.448,55.108,159.801
C08583=1017.182,-81.199,-100.246,165.444,55.115,159.802
C08584=1017.177,-81.449,-100.237,165.442,55.120,159.802
C08585=1017.171,-81.698,-100.227,165.439,55.126,159.802
C08586=1017.167,-81.948,-100.218,165.436,55.133,159.803
C08587=1017.161,-82.198,-100.209,165.433,55.138,159.803
C08588=1017.155,-82.448,-100.200,165.430,55.144,159.804
C08589=1017.150,-82.697,-100.190,165.427,55.151,159.804
C08590=1017.145,-82.947,-100.182,165.424,55.156,159.804
C08591=1017.140,-83.197,-100.171,165.421,55.162,159.805
C08592=1017.135,-83.447,-100.163,165.418,55.169,159.805
C08593=1017.130,-83.696,-100.153,165.415,55.174,159.806
C08594=1017.124,-83.947,-100.144,165.412,55.180,159.806
C08595=1017.119,-84.197,-100.135,165.408,55.186,159.806
C08596=1017.114,-84.446,-100.126,165.406,55.192,159.807
C08597=1017.108,-84.696,-100.118,165.403,55.198,159.807
C08598=1017.103,-84.946,-100.107,165.400,55.204,159.807
C08599=1017.098,-85.195,-100.099,165.397,55.210,159.808
C08600=1017.092,-85.476,-100.088,165.393,55.216,159.808
C08601=1017.086,-85.757,-100.078,165.390,55.223,159.809
C08602=1017.080,-86.037,-100.068,165.387,55.230,159.809
C08603=1017.075,-86.318,-100.058,165.383,55.237,159.810
C08604=1017.069,-86.567,-100.049,165.381,55.242,159.810
C08605=1017.065,-86.817,-100.040,165.377,55.249,159.810
C08606=1017.059,-87.067,-100.030,165.375,55.255,159.811
C08607=1017.053,-87.317,-100.021,165.372,55.260,159.811
C08608=1017.049,-87.567,-100.012,165.368,55.266,159.811
C08609=1017.043,-87.816,-100.003,165.366,55.273,159.812
C08610=1017.038,-88.067,-99.994,165.363,55.278,159.812
C08611=1017.033,-88.316,-99.985,165.359,55.284,159.813
C08612=1017.027,-88.565,-99.976,165.356,55.290,159.813
C08613=1017.023,-88.815,-99.967,165.354,55.296,159.813
C08614=1017.017,-89.065,-99.958,165.351,55.301,159.814
C08615=1017.012,-89.315,-99.948,165.348,55.308,159.814
C08616=1017.007,-89.565,-99.940,165.345,55.314,159.814
C08617=1017.002,-89.815,-99.931,165.342,55.319,159.815
C08618=1016.997,-90.064,-99.922,165.338,55.325,159.815
C08619=1016.991,-90.314,-99.913,165.335,55.331,159.815
C08620=1016.987,-90.564,-99.904,165.333,55.337,159.816
C08621=1016.982,-90.814,-99.895,165.330,55.343,159.816
C08622=1016.976,-91.064,-99.885,165.327,55.349,159.817
C08623=1016.971,-91.313,-99.877,165.324,55.355,159.817
C08624=1016.966,-91.563,-99.868,165.321,55.360,159.817
C08625=1016.961,-91.813,-99.859,165.318,55.366,159.818
C08626=1016.955,-92.062,-99.850,165.315,55.372,159.818
C08627=1016.951,-92.312,-99.841,165.312,55.378,159.818
C08628=1016.946,-92.562,-99.833,165.309,55.383,159.819
C08629=1016.940,-92.812,-99.824,165.306,55.389,159.819
C08630=1016.936,-93.062,-99.815,165.302,55.395,159.819
C08631=1016.930,-93.312,-99.805,165.300,55.402,159.820
C08632=1016.925,-93.562,-99.796,165.297,55.407,159.820
C08633=1016.920,-93.811,-99.788,165.295,55.413,159.820
C08634=1016.915,-94.061,-99.779,165.291,55.419,159.821
C08635=1016.910,-94.311,-99.770,165.288,55.425,159.821
C08636=1016.905,-94.561,-99.762,165.285,55.430,159.821
C08637=1016.900,-94.810,-99.752,165.283,55.436,159.822
C08638=1016.895,-95.060,-99.743,165.279,55.442,159.822
C08639=1016.890,-95.310,-99.735,165.276,55.448,159.822
C08640=1016.885,-95.560,-99.726,165.273,55.453,159.823
C08641=1016.880,-95.809,-99.717,165.271,55.459,159.823
C08642=1016.875,-96.059,-99.708,165.268,55.465,159.823
C08643=1016.870,-96.309,-99.700,165.264,55.471,159.824
C08644=1016.865,-96.559,-99.691,165.261,55.476,159.824
C08645=1016.860,-96.809,-99.682,165.259,55.482,159.824
C08646=1016.855,-97.059,-99.674,165.256,55.488,159.825
C08647=1016.850,-97.308,-99.664,165.253,55.493,159.825
C08648=1016.845,-97.558,-99.656,165.249,55.499,159.825
C08649=1016.840,-97.807,-99.647,165.247,55.505,159.826
C08650=1016.835,-98.058,-99.639,165.244,55.511,159.826
C08651=1016.830,-98.308,-99.630,165.241,55.516,159.826
C08652=1016.825,-98.557,-99.622,165.237,55.522,159.827
C08653=1016.820,-98.807,-99.613,165.234,55.528,159.827
C08654=1016.814,-99.057,-99.605,165.232,55.534,159.827
C08655=1016.809,-99.307,-99.596,165.228,55.541,159.828
C08656=1016.804,-99.556,-99.588,165.226,55.546,159.828
C08657=1016.798,-99.806,-99.579,165.223,55.552,159.828
C08658=1016.794,-100.056,-99.570,165.220,55.558,159.829
C08659=1016.789,-100.306,-99.562,165.216,55.564,159.829
C08660=1016.784,-100.556,-99.554,165.214,55.569,159.829
C08661=1016.778,-100.806,-99.545,165.211,55.576,159.830
C08662=1016.773,-101.056,-99.537,165.208,55.582,159.830
C08663=1016.769,-101.305,-99.529,165.205,55.587,159.830
C08664=1016.763,-101.588,-99.519,165.202,55.594,159.831
C08665=1016.756,-101.871,-99.510,165.198,55.600,159.831
C08666=1016.751,-102.153,-99.501,165.195,55.607,159.832
C08667=1016.746,-102.436,-99.491,165.191,55.614,159.832
C08668=1016.740,-102.686,-99.483,165.189,55.620,159.832
C08669=1016.735,-102.936,-99.474,165.186,55.625,159.833
C08670=1016.730,-103.185,-99.466,165.183,55.631,159.833
C08671=1016.726,-103.435,-99.458,165.179,55.637,159.833
C08672=1016.720,-103.685,-99.450,165.177,55.643,159.834
C08673=1016.715,-103.934,-99.441,165.174,55.648,159.834
C08674=1016.710,-104.185,-99.433,165.171,55.654,159.834
C08675=1016.705,-104.434,-99.425,165.167,55.660,159.834
C08676=1016.700,-104.684,-99.416,165.165,55.666,159.835
C08677=1016.695,-104.934,-99.407,165.162,55.672,159.835
C08678=1016.691,-105.184,-99.400,165.159,55.677,159.836
C08679=1016.685,-105.434,-99.391,165.155,55.683,159.836
C08680=1016.680,-105.683,-99.383,165.153,55.689,159.836
C08681=1016.675,-105.934,-99.375,165.150,55.695,159.836
C08682=1016.670,-106.183,-99.367,165.148,55.701,159.837
C08683=1016.666,-106.433,-99.359,165.144,55.707,159.837
C08684=1016.660,-106.683,-99.351,165.141,55.713,159.838
C08685=1016.655,-106.932,-99.342,165.138,55.719,159.838
C08686=1016.650,-107.183,-99.335,165.136,55.724,159.838
C08687=1016.645,-107.432,-99.326,165.133,55.730,159.839
C08688=1016.640,-107.681,-99.318,165.129,55.736,159.839
C08689=1016.635,-107.932,-99.310,165.126,55.742,159.839
C08690=1016.630,-108.181,-99.302,165.124,55.748,159.840
C08691=1016.625,-108.432,-99.294,165.121,55.753,159.840
C08692=1016.620,-108.681,-99.286,165.117,55.759,159.840
C08693=1016.615,-108.931,-99.278,165.115,55.765,159.840
C08694=1016.609,-109.181,-99.270,165.112,55.771,159.841
C08695=1016.604,-109.431,-99.262,165.108,55.777,159.841
C08696=1016.600,-109.681,-99.255,165.105,55.782,159.841
C08697=1016.595,-109.930,-99.247,165.103,55.788,159.842
C08698=1016.590,-110.181,-99.239,165.100,55.794,159.842
C08699=1016.585,-110.430,-99.231,165.096,55.800,159.842
C08700=1016.580,-110.680,-99.223,165.093,55.806,159.843
C08701=1016.575,-110.930,-99.214,165.091,55.812,159.843
C08702=1016.570,-111.180,-99.207,165.088,55.818,159.844
C08703=1016.565,-111.429,-99.199,165.085,55.824,159.844
C08704=1016.560,-111.679,-99.191,165.082,55.830,159.844
C08705=1016.555,-111.929,-99.184,165.079,55.835,159.844
C08706=1016.550,-112.178,-99.175,165.077,55.841,159.845
C08707=1016.545,-112.429,-99.168,165.074,55.847,159.845
C08708=1016.540,-112.678,-99.159,165.070,55.853,159.845
C08709=1016.535,-112.928,-99.152,165.067,55.859,159.846
C08710=1016.530,-113.178,-99.144,165.065,55.864,159.846
C08711=1016.525,-113.427,-99.136,165.062,55.870,159.846
C08712=1016.520,-113.677,-99.129,165.059,55.875,159.846
C08713=1016.515,-113.928,-99.121,165.055,55.881,159.847
C08714=1016.510,-114.177,-99.113,165.052,55.887,159.847
C08715=1016.506,-114.427,-99.105,165.049,55.892,159.847
C08716=1016.501,-114.677,-99.097,165.047,55.898,159.848
C08717=1016.496,-114.926,-99.089,165.044,55.904,159.848
C08718=1016.490,-115.176,-99.082,165.040,55.910,159.848
C08719=1016.486,-115.426,-99.075,165.038,55.916,159.849
C08720=1016.481,-115.676,-99.067,165.035,55.921,159.849
C08721=1016.476,-115.927,-99.059,165.032,55.927,159.849
C08722=1016.471,-116.175,-99.052,165.028,55.933,159.849
C08723=1016.466,-116.426,-99.044,165.026,55.939,159.850
C08724=1016.461,-116.675,-99.036,165.023,55.945,159.850
C08725=1016.456,-116.926,-99.029,165.020,55.950,159.851
C08726=1016.451,-117.175,-99.022,165.018,55.956,159.851
C08727=1016.446,-117.425,-99.013,165.014,55.962,159.851
C08728=1016.440,-117.708,-99.005,165.011,55.969,159.851
C08729=1016.435,-117.991,-98.996,165.008,55.976,159.852
C08730=1016.430,-118.273,-98.988,165.005,55.982,159.852
C08731=1016.424,-118.556,-98.979,165.001,55.988,159.853
C08732=1016.419,-118.807,-98.972,164.999,55.994,159.853
C08733=1016.414,-119.056,-98.964,164.995,56.000,159.853
C08734=1016.409,-119.306,-98.957,164.992,56.006,159.854
C08735=1016.404,-119.555,-98.949,164.989,56.012,159.854
C08736=1016.399,-119.806,-98.941,164.987,56.018,159.854
C08737=1016.394,-120.055,-98.934,164.984,56.023,159.855
C08738=1016.389,-120.305,-98.927,164.980,56.029,159.855
C08739=1016.385,-120.555,-98.919,164.978,56.035,159.855
C08740=1016.379,-120.805,-98.912,164.974,56.040,159.855
C08741=1016.375,-121.055,-98.905,164.972,56.046,159.856
C08742=1016.370,-121.304,-98.897,164.969,56.052,159.856
C08743=1016.365,-121.554,-98.890,164.966,56.057,159.856
C08744=1016.360,-121.804,-98.883,164.963,56.063,159.856
C08745=1016.355,-122.054,-98.875,164.960,56.069,159.857
C08746=1016.350,-122.304,-98.868,164.957,56.075,159.857
C08747=1016.345,-122.554,-98.860,164.954,56.081,159.857
C08748=1016.341,-122.804,-98.853,164.952,56.086,159.858
C08749=1016.335,-123.054,-98.846,164.949,56.092,159.858
C08750=1016.331,-123.303,-98.838,164.945,56.098,159.858
C08751=1016.326,-123.553,-98.831,164.943,56.104,159.859
C08752=1016.321,-123.803,-98.824,164.939,56.109,159.859
C08753=1016.316,-124.052,-98.816,164.937,56.115,159.859
C08754=1016.311,-124.303,-98.809,164.934,56.120,159.859
C08755=1016.306,-124.552,-98.802,164.931,56.126,159.860
C08756=1016.302,-124.802,-98.795,164.929,56.132,159.860
C08757=1016.297,-125.052,-98.788,164.925,56.138,159.860
C08758=1016.292,-125.302,-98.781,164.922,56.144,159.861
C08759=1016.287,-125.552,-98.773,164.919,56.149,159.861
C08760=1016.282,-125.802,-98.766,164.917,56.155,159.861
C08761=1016.277,-126.051,-98.759,164.914,56.161,159.862
C08762=1016.272,-126.302,-98.752,164.910,56.167,159.862
C08763=1016.267,-126.551,-98.745,164.908,56.173,159.862
C08764=1016.263,-126.801,-98.738,164.905,56.178,159.863
C08765=1016.257,-127.051,-98.731,164.902,56.183,159.863
C08766=1016.253,-127.301,-98.723,164.899,56.189,159.863
C08767=1016.248,-127.551,-98.717,164.896,56.195,159.863
C08768=1016.244,-127.800,-98.710,164.894,56.201,159.864
C08769=1016.239,-128.049,-98.703,164.890,56.207,159.864
C08770=1016.234,-128.300,-98.695,164.887,56.213,159.864
C08771=1016.229,-128.549,-98.687,164.885,56.217,159.865
C08772=1016.225,-128.799,-98.679,164.882,56.221,159.865
C08773=1016.222,-129.048,-98.670,164.880,56.225,159.865
C08774=1016.219,-129.298,-98.661,164.877,56.228,159.864
C08775=1016.216,-129.547,-98.650,164.874,56.231,159.864
C08776=1016.214,-129.797,-98.639,164.872,56.233,159.864
C08777=1016.212,-130.047,-98.627,164.869,56.235,159.864
C08778=1016.211,-130.297,-98.616,164.867,56.235,159.863
C08779=1016.209,-130.546,-98.603,164.864,56.236,159.863
C08780=1016.209,-130.796,-98.590,164.862,56.236,159.862
C08781=1016.208,-131.045,-98.576,164.859,56.234,159.861
C08782=1016.209,-131.295,-98.561,164.857,56.233,159.860
C08783=1016.209,-131.545,-98.546,164.856,56.231,159.860
C08784=1016.209,-131.795,-98.531,164.854,56.229,159.859
C08785=1016.210,-132.045,-98.514,164.852,56.226,159.858
C08786=1016.212,-132.294,-98.497,164.849,56.222,159.856
C08787=1016.214,-132.543,-98.480,164.848,56.218,159.855
C08788=1016.217,-132.793,-98.462,164.846,56.213,159.854
C08789=1016.220,-133.043,-98.444,164.844,56.208,159.853
C08790=1016.222,-133.292,-98.424,164.843,56.202,159.851
C08791=1016.225,-133.542,-98.405,164.841,56.196,159.850
C08792=1015.975,-133.568,-98.798,164.804,56.563,159.905
C08793=1015.972,-133.319,-98.818,164.806,56.569,159.907
C08794=1015.969,-133.069,-98.838,164.807,56.576,159.908
C08795=1015.966,-132.819,-98.857,164.808,56.581,159.910
C08796=1015.964,-132.570,-98.875,164.811,56.586,159.911
C08797=1015.962,-132.320,-98.892,164.812,56.590,159.912
C08798=1015.960,-132.071,-98.909,164.815,56.594,159.914
C08799=1015.959,-131.821,-98.925,164.817,56.597,159.915
C08800=1015.958,-131.571,-98.941,164.819,56.599,159.916
C08801=1015.958,-131.321,-98.956,164.821,56.601,159.916
C08802=1015.958,-131.071,-98.970,164.823,56.602,159.917
C08803=1015.959,-130.822,-98.985,164.825,56.603,159.918
C08804=1015.960,-130.573,-98.998,164.828,56.603,159.919
C08805=1015.960,-130.322,-99.010,164.830,56.602,159.919
C08806=1015.962,-130.073,-99.023,164.832,56.601,159.919
C08807=1015.964,-129.823,-99.034,164.835,56.600,159.920
C08808=1015.966,-129.574,-99.045,164.838,56.598,159.920
C08809=1015.968,-129.324,-99.055,164.840,56.596,159.920
C08810=1015.972,-129.075,-99.065,164.843,56.592,159.921
C08811=1015.975,-128.825,-99.074,164.846,56.589,159.921
C08812=1015.978,-128.575,-99.082,164.848,56.584,159.920
C08813=1015.983,-128.326,-99.090,164.850,56.579,159.920
C08814=1015.987,-128.076,-99.098,164.853,56.574,159.920
C08815=1015.993,-127.827,-99.105,164.857,56.568,159.920
C08816=1015.997,-127.577,-99.111,164.859,56.562,159.919
C08817=1016.002,-127.327,-99.118,164.862,56.556,159.919
C08818=1016.007,-127.077,-99.126,164.865,56.551,159.919
C08819=1016.012,-126.828,-99.133,164.867,56.545,159.918
C08820=1016.016,-126.577,-99.140,164.871,56.539,159.918
C08821=1016.021,-126.328,-99.147,164.874,56.533,159.918
C08822=1016.026,-126.078,-99.154,164.876,56.527,159.918
C08823=1016.032,-125.828,-99.161,164.879,56.521,159.917
C08824=1016.036,-125.578,-99.168,164.882,56.516,159.917
C08825=1016.041,-125.328,-99.175,164.885,56.510,159.917
C08826=1016.046,-125.078,-99.182,164.888,56.504,159.916
C08827=1016.051,-124.829,-99.189,164.891,56.498,159.916
C08828=1016.055,-124.579,-99.197,164.893,56.492,159.916
C08829=1016.061,-124.329,-99.204,164.896,56.486,159.915
C08830=1016.065,-124.079,-99.210,164.900,56.480,159.915
C08831=1016.069,-123.829,-99.218,164.903,56.475,159.915
C08832=1016.075,-123.579,-99.225,164.905,56.469,159.915
C08833=1016.079,-123.330,-99.232,164.908,56.464,159.914
C08834=1016.084,-123.079,-99.240,164.911,56.458,159.914
C08835=1016.089,-122.830,-99.247,164.914,56.452,159.914
C08836=1016.094,-122.580,-99.254,164.917,56.446,159.913
C08837=1016.099,-122.330,-99.262,164.920,56.440,159.913
C08838=1016.104,-122.081,-99.269,164.922,56.434,159.913
C08839=1016.109,-121.830,-99.277,164.925,56.429,159.912
C08840=1016.114,-121.581,-99.284,164.929,56.423,159.912
C08841=1016.118,-121.331,-99.291,164.931,56.417,159.912
C08842=1016.123,-121.081,-99.299,164.934,56.411,159.911
C08843=1016.127,-120.831,-99.306,164.937,56.405,159.911
C08844=1016.133,-120.581,-99.313,164.939,56.400,159.911
C08845=1016.138,-120.332,-99.321,164.943,56.393,159.911
C08846=1016.142,-120.081,-99.328,164.946,56.388,159.910
C08847=1016.148,-119.832,-99.335,164.948,56.382,159.910
C08848=1016.153,-119.582,-99.343,164.951,56.376,159.909
C08849=1016.157,-119.332,-99.350,164.955,56.370,159.909
C08850=1016.162,-119.083,-99.357,164.957,56.364,159.909
C08851=1016.167,-118.832,-99.365,164.960,56.358,159.909
C08852=1016.171,-118.583,-99.372,164.963,56.353,159.908
C08853=1016.177,-118.300,-99.381,164.966,56.347,159.908
C08854=1016.183,-118.017,-99.390,164.970,56.340,159.908
C08855=1016.188,-117.735,-99.397,164.973,56.333,159.907
C08856=1016.194,-117.452,-99.407,164.976,56.326,159.907
C08857=1016.199,-117.203,-99.414,164.979,56.320,159.906
C08858=1016.204,-116.952,-99.422,164.982,56.314,159.906
C08859=1016.209,-116.702,-99.429,164.985,56.308,159.906
C08860=1016.213,-116.452,-99.437,164.988,56.302,159.905
C08861=1016.219,-116.202,-99.444,164.990,56.297,159.905
C08862=1016.223,-115.953,-99.452,164.994,56.290,159.905
C08863=1016.228,-115.703,-99.460,164.997,56.285,159.905
C08864=1016.233,-115.453,-99.467,164.999,56.279,159.904
C08865=1016.238,-115.203,-99.474,165.002,56.273,159.904
C08866=1016.243,-114.954,-99.482,165.006,56.267,159.904
C08867=1016.248,-114.704,-99.490,165.008,56.261,159.903
C08868=1016.253,-114.454,-99.498,165.011,56.256,159.903
C08869=1016.257,-114.204,-99.505,165.014,56.250,159.903
C08870=1016.263,-113.954,-99.513,165.017,56.244,159.902
C08871=1016.268,-113.705,-99.521,165.020,56.238,159.902
C08872=1016.273,-113.455,-99.528,165.023,56.232,159.902
C08873=1016.278,-113.204,-99.536,165.025,56.227,159.901
C08874=1016.282,-112.955,-99.544,165.029,56.220,159.901
C08875=1016.287,-112.705,-99.552,165.032,56.215,159.901
C08876=1016.292,-112.455,-99.560,165.035,56.209,159.900
C08877=1016.297,-112.206,-99.568,165.038,56.203,159.900
C08878=1016.303,-111.956,-99.575,165.041,56.197,159.900
C08879=1016.307,-111.706,-99.583,165.044,56.191,159.900
C08880=1016.312,-111.456,-99.591,165.046,56.186,159.899
C08881=1016.317,-111.206,-99.599,165.049,56.179,159.899
C08882=1016.322,-110.957,-99.607,165.052,56.173,159.898
C08883=1016.327,-110.706,-99.615,165.055,56.167,159.898
C08884=1016.332,-110.456,-99.622,165.059,56.161,159.898
C08885=1016.336,-110.207,-99.631,165.061,56.155,159.897
C08886=1016.342,-109.957,-99.638,165.064,56.150,159.897
C08887=1016.347,-109.707,-99.646,165.067,56.144,159.897
C08888=1016.352,-109.458,-99.654,165.070,56.138,159.897
C08889=1016.357,-109.207,-99.661,165.073,56.132,159.896
C08890=1016.362,-108.958,-99.670,165.075,56.126,159.896
C08891=1016.366,-108.708,-99.677,165.079,56.119,159.895
C08892=1016.372,-108.458,-99.686,165.081,56.114,159.895
C08893=1016.377,-108.208,-99.694,165.084,56.108,159.895
C08894=1016.382,-107.958,-99.702,165.088,56.102,159.895
C08895=1016.386,-107.709,-99.709,165.091,56.096,159.894
C08896=1016.391,-107.459,-99.718,165.093,56.090,159.894
C08897=1016.396,-107.209,-99.726,165.097,56.084,159.894
C08898=1016.402,-106.959,-99.734,165.100,56.078,159.893
C08899=1016.406,-106.709,-99.742,165.102,56.072,159.893
C08900=1016.411,-106.460,-99.750,165.105,56.066,159.892
C08901=1016.417,-106.210,-99.759,165.108,56.060,159.892
C08902=1016.422,-105.960,-99.766,165.111,56.054,159.892
C08903=1016.426,-105.711,-99.774,165.114,56.049,159.891
C08904=1016.431,-105.460,-99.782,165.117,56.043,159.891
C08905=1016.436,-105.210,-99.791,165.120,56.037,159.891
C08906=1016.442,-104.961,-99.799,165.123,56.031,159.890
C08907=1016.447,-104.710,-99.807,165.126,56.025,159.890
C08908=1016.451,-104.461,-99.815,165.129,56.019,159.890
C08909=1016.457,-104.212,-99.824,165.131,56.013,159.889
C08910=1016.462,-103.961,-99.831,165.134,56.007,159.889
C08911=1016.467,-103.712,-99.840,165.138,56.001,159.889
C08912=1016.472,-103.462,-99.848,165.140,55.995,159.888
C08913=1016.476,-103.212,-99.856,165.143,55.990,159.888
C08914=1016.481,-102.962,-99.865,165.147,55.983,159.888
C08915=1016.486,-102.713,-99.873,165.150,55.978,159.887
C08916=1016.491,-102.463,-99.882,165.152,55.972,159.887
C08917=1016.498,-102.180,-99.891,165.155,55.965,159.887
C08918=1016.503,-101.898,-99.900,165.159,55.958,159.886
C08919=1016.508,-101.615,-99.910,165.162,55.952,159.886
C08920=1016.514,-101.332,-99.919,165.165,55.945,159.885
C08921=1016.520,-101.082,-99.927,165.169,55.939,159.885
C08922=1016.524,-100.832,-99.936,165.172,55.933,159.885
C08923=1016.529,-100.583,-99.944,165.174,55.927,159.884
C08924=1016.534,-100.333,-99.952,165.178,55.920,159.884
C08925=1016.539,-100.083,-99.961,165.180,55.915,159.884
C08926=1016.544,-99.834,-99.969,165.184,55.908,159.883
C08927=1016.550,-99.584,-99.978,165.187,55.903,159.883
C08928=1016.555,-99.334,-99.986,165.189,55.897,159.883
C08929=1016.560,-99.085,-99.995,165.193,55.890,159.882
C08930=1016.565,-98.834,-100.002,165.195,55.885,159.882
C08931=1016.570,-98.584,-100.011,165.198,55.879,159.881
C08932=1016.575,-98.334,-100.020,165.202,55.873,159.881
C08933=1016.580,-98.085,-100.028,165.204,55.866,159.881
C08934=1016.585,-97.835,-100.037,165.207,55.861,159.880
C08935=1016.591,-97.585,-100.045,165.210,55.854,159.880
C08936=1016.595,-97.335,-100.054,165.213,55.849,159.880
C08937=1016.600,-97.086,-100.063,165.216,55.843,159.879
C08938=1016.605,-96.836,-100.072,165.218,55.837,159.879
C08939=1016.610,-96.586,-100.080,165.222,55.831,159.879
C08940=1016.616,-96.336,-100.089,165.225,55.826,159.878
C08941=1016.620,-96.086,-100.098,165.228,55.820,159.878
C08942=1016.625,-95.837,-100.106,165.231,55.814,159.878
C08943=1016.629,-95.587,-100.115,165.234,55.808,159.877
C08944=1016.634,-95.337,-100.124,165.237,55.802,159.877
C08945=1016.640,-95.088,-100.132,165.239,55.796,159.876
C08946=1016.645,-94.837,-100.142,165.243,55.790,159.876
C08947=1016.650,-94.587,-100.150,165.245,55.784,159.876
C08948=1016.656,-94.338,-100.159,165.248,55.778,159.876
C08949=1016.660,-94.088,-100.168,165.252,55.772,159.875
C08950=1016.666,-93.838,-100.177,165.255,55.767,159.875
C08951=1016.670,-93.588,-100.186,165.257,55.761,159.875
C08952=1016.675,-93.339,-100.194,165.260,55.755,159.874
